KUKA KRL program: EPS_2_251245_SANMH3A_A_20250910013112.src

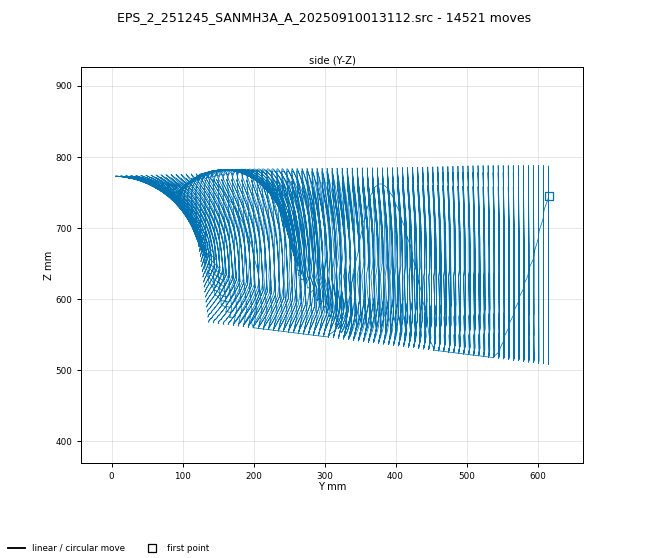
[picture p0: tool path of EPS_2_251245_SANMH3A_A_20250910013112.src, 14521 of 14523 moves have a stored position in this frame; points joined in program order, loops and branches not executed]
&ACCESS RVP
&REL 4
&COMMENT QRS 19112012
&PARAM EDITMASK = *
DEF PART()
EXT BAS (BAS_COMMAND :IN,REAL :IN )
INT I
BAS (#INITMOV,0 )

;KUKA QRS Post kuka4.cps  Date:22-06-2017 !

File_ID=2817

QRS_PRE_INIT()

;Init var - Until changes are made in qrs_pre_init
Outlet_Square_prg=0
Inlet_1_Square_prg=0
Inlet_2_Square_prg=0
Inlet_3_Square_prg=0
Inlet_4_Square_prg=0
Inlet_5_Square_prg=0

Outlet_1={X 0.000, Y 519.160, Z 687.500, B 0.000, E1 0.000 }
Inlet_1={X 0.000, Y 520.240, Z 710.500, B 0.000, E1 90.000 }
Inlet_2={X 0.000, Y 521.300, Z 657.500, B 0.000, E1 180.000 }
Outlet_1_type=201
Inlet_1_type=135
Inlet_2_type=201
;QRS#1=Sidecore dimensions
;QRS#2=200-8" PVC SDR 35
;QRS#3=135-5" PVC SDR 28
;QRS#4=200-8" PVC SDR 35
;QRS#5=
;QRS#6=
;QRS#7=
;QRS#8=
;QRS#9=12-08 PSX
;QRS#10=8-11 PSX
;QRS#11=12-08 PSX
;QRS#12=
;QRS#13=
;QRS#14=
;QRS#15=
;QRS#16=1220x127x1067 3,5'
;QRS#17=EPS Height
;QRS#18=788
;QRS#19=*
;QRS#20= UPDATED VERSION 22-06-2017
;QRS#21=*
Outlet_Square=0100
Inlet_1_Square=070
Inlet_2_Square=0100
Inlet_3_Square=0
Inlet_4_Square=0
Inlet_5_Square=0
Mill_Square=1
Outlet_Square_Prg=204
Inlet_1_Square_prg=202
Inlet_2_Square_prg=204

QRS_INIT()

$ADVANCE=5

; T1
PTP {E1 173.419,E2 173.419}
PTP {X 0,Y 615.493,A -85,B 0,C 180,E1 173.419,E2 173.419,E3 0,E4 0,E5 0,E6 0}
QRS_SPEED_INIT()
LIN {X 0,Y 615.493,Z 745.39,A -85,B 0,C 180,E1 173.419,E2 173.419,E3 0,E4 0,E5 0,E6 0} C_VEL
LIN {X 0,Y 615.498,Z 736.605,A -85,B 0,C 180,E1 172.784,E2 172.784} C_VEL
LIN {X 0,Y 615.5,Z 727.686,A -85,B 0,C 180,E1 172.29,E2 172.29} C_VEL
LIN {X 0,Y 615.493,Z 717.685,A -85,B 0,C 180,E1 171.877,E2 171.877} C_VEL
LIN {X 0,Y 615.488,Z 709.508,A -85,B 0,C 180,E1 171.629,E2 171.629} C_VEL
LIN {X 0,Y 615.491,Z 700.427,A -85,B 0,C 180,E1 171.443,E2 171.443} C_VEL
LIN {X 0,Y 615.487,Z 631.25,A -85,B 0,C 180,E1 170.615,E2 170.615} C_VEL
LIN {X 0,Y 615.498,Z 629.569,A -85,B 0,C 180,E1 170.47,E2 170.47} C_VEL
LIN {X 0,Y 615.491,Z 604.096,A -85,B 0,C 180,E1 167.47,E2 167.47} C_VEL
LIN {X 0,Y 615.496,Z 580.016,A -85,B 0,C 180,E1 164.605,E2 164.605} C_VEL
LIN {X 0,Y 615.48,Z 556.069,A -85,B 0,C 180,E1 161.719,E2 161.719} C_VEL
LIN {X 0,Y 615.495,Z 533.177,A -85,B 0,C 180,E1 158.919,E2 158.919} C_VEL
LIN {X 0,Y 615.496,Z 511.475,A -85,B 0,C 180,E1 156.217,E2 156.217} C_VEL
LIN {X 0,Y 615.495,Z 507.92,A -85,B 0,C 180,E1 155.728,E2 155.728} C_VEL
LIN {X 0,Y 615.497,Z 507.698,A -85,B 0,C 180,E1 153.556,E2 153.556} C_VEL
LIN {X 0,Y 615.49,Z 507.693,A -85,B 0,C 180,E1 151.342,E2 151.342} C_VEL
LIN {X 0,Y 615.477,Z 507.686,A -85,B 0,C 180,E1 148.916,E2 148.916} C_VEL
LIN {X 0,Y 615.485,Z 507.682,A -85,B 0,C 180,E1 146.467,E2 146.467} C_VEL
LIN {X 0,Y 615.489,Z 507.701,A -85,B 0,C 180,E1 143.575,E2 143.575} C_VEL
LIN {X 0,Y 615.479,Z 507.687,A -85,B 0,C 180,E1 140.939,E2 140.939} C_VEL
LIN {X 0,Y 615.482,Z 507.683,A -85,B 0,C 180,E1 138.525,E2 138.525} C_VEL
LIN {X 0,Y 615.485,Z 507.691,A -85,B 0,C 180,E1 135.85,E2 135.85} C_VEL
LIN {X 0,Y 615.485,Z 507.689,A -85,B 0,C 180,E1 133.047,E2 133.047} C_VEL
LIN {X 0,Y 615.478,Z 507.684,A -85,B 0,C 180,E1 130.608,E2 130.608} C_VEL
LIN {X 0,Y 615.489,Z 507.685,A -85,B 0,C 180,E1 128.012,E2 128.012} C_VEL
LIN {X 0,Y 615.488,Z 507.695,A -85,B 0,C 180,E1 125.616,E2 125.616} C_VEL
LIN {X 0,Y 615.492,Z 507.696,A -85,B 0,C 180,E1 123.236,E2 123.236} C_VEL
LIN {X 0,Y 615.479,Z 507.69,A -85,B 0,C 180,E1 120.921,E2 120.921} C_VEL
LIN {X 0,Y 615.481,Z 507.683,A -85,B 0,C 180,E1 118.449,E2 118.449} C_VEL
LIN {X 0,Y 615.484,Z 507.69,A -85,B 0,C 180,E1 115.716,E2 115.716} C_VEL
LIN {X 0,Y 615.48,Z 507.689,A -85,B 0,C 180,E1 112.845,E2 112.845} C_VEL
LIN {X 0,Y 615.493,Z 507.682,A -85,B 0,C 180,E1 110.033,E2 110.033} C_VEL
LIN {X 0,Y 615.498,Z 507.867,A -85,B 0,C 180,E1 109.208,E2 109.208} C_VEL
LIN {X 0,Y 615.49,Z 524.635,A -85,B 0,C 180,E1 106.431,E2 106.431} C_VEL
LIN {X 0,Y 615.487,Z 541.428,A -85,B 0,C 180,E1 103.706,E2 103.706} C_VEL
LIN {X 0,Y 615.484,Z 547.062,A -85,B 0,C 180,E1 102.845,E2 102.845} C_VEL
LIN {X 0,Y 615.481,Z 549.379,A -85,B 0,C 180,E1 102.782,E2 102.782} C_VEL
LIN {X 0,Y 615.497,Z 653.612,A -85,B 0,C 180,E1 101.548,E2 101.548} C_VEL
LIN {X 0,Y 615.498,Z 666.203,A -85,B 0,C 180,E1 101.277,E2 101.277} C_VEL
LIN {X 0,Y 615.497,Z 679.523,A -85,B 0,C 180,E1 100.845,E2 100.845} C_VEL
LIN {X 0,Y 615.495,Z 690.554,A -85,B 0,C 180,E1 100.361,E2 100.361} C_VEL
LIN {X 0,Y 615.489,Z 702.297,A -85,B 0,C 180,E1 99.697,E2 99.697} C_VEL
LIN {X 0,Y 615.499,Z 712.761,A -85,B 0,C 180,E1 98.951,E2 98.951} C_VEL
LIN {X 0,Y 615.498,Z 721.325,A -85,B 0,C 180,E1 98.206,E2 98.206} C_VEL
LIN {X 0,Y 615.497,Z 729.204,A -85,B 0,C 180,E1 97.381,E2 97.381} C_VEL
LIN {X 0,Y 615.497,Z 736.895,A -85,B 0,C 180,E1 96.393,E2 96.393} C_VEL
LIN {X 0,Y 615.497,Z 743.955,A -85,B 0,C 180,E1 95.242,E2 95.242} C_VEL
LIN {X 0,Y 615.494,Z 748.655,A -85,B 0,C 180,E1 94.257,E2 94.257} C_VEL
LIN {X 0,Y 615.494,Z 752.253,A -85,B 0,C 180,E1 93.273,E2 93.273} C_VEL
LIN {X 0,Y 615.496,Z 754.113,A -85,B 0,C 180,E1 92.618,E2 92.618} C_VEL
LIN {X 0,Y 615.498,Z 755.532,A -85,B 0,C 180,E1 91.964,E2 91.964} C_VEL
LIN {X 0,Y 615.496,Z 757.141,A -85,B 0,C 180,E1 90.655,E2 90.655} C_VEL
LIN {X 0,Y 615.495,Z 757.384,A -85,B 0,C 180,E1 90.001,E2 90.001} C_VEL
LIN {X 0,Y 615.495,Z 757.206,A -85,B 0,C 180,E1 89.346,E2 89.346} C_VEL
LIN {X 0,Y 615.499,Z 755.683,A -85,B 0,C 180,E1 88.038,E2 88.038} C_VEL
LIN {X 0,Y 615.498,Z 754.343,A -85,B 0,C 180,E1 87.383,E2 87.383} C_VEL
LIN {X 0,Y 615.496,Z 751.496,A -85,B 0,C 180,E1 86.4,E2 86.4} C_VEL
LIN {X 0,Y 615.498,Z 747.637,A -85,B 0,C 180,E1 85.416,E2 85.416} C_VEL
LIN {X 0,Y 615.498,Z 742.655,A -85,B 0,C 180,E1 84.431,E2 84.431} C_VEL
LIN {X 0,Y 615.496,Z 736.208,A -85,B 0,C 180,E1 83.418,E2 83.418} C_VEL
LIN {X 0,Y 615.497,Z 728.543,A -85,B 0,C 180,E1 82.455,E2 82.455} C_VEL
LIN {X 0,Y 615.498,Z 718.766,A -85,B 0,C 180,E1 81.464,E2 81.464} C_VEL
LIN {X 0,Y 615.498,Z 708.502,A -85,B 0,C 180,E1 80.636,E2 80.636} C_VEL
LIN {X 0,Y 615.495,Z 696.941,A -85,B 0,C 180,E1 79.889,E2 79.889} C_VEL
LIN {X 0,Y 615.497,Z 685.031,A -85,B 0,C 180,E1 79.291,E2 79.291} C_VEL
LIN {X 0,Y 615.497,Z 672.179,A -85,B 0,C 180,E1 78.808,E2 78.808} C_VEL
LIN {X 0,Y 615.497,Z 659.587,A -85,B 0,C 180,E1 78.474,E2 78.474} C_VEL
LIN {X 0,Y 615.498,Z 646.491,A -85,B 0,C 180,E1 78.265,E2 78.265} C_VEL
LIN {X 0,Y 615.487,Z 547.562,A -85,B 0,C 180,E1 77.093,E2 77.093} C_VEL
LIN {X 0,Y 615.486,Z 546.205,A -85,B 0,C 180,E1 76.967,E2 76.967} C_VEL
LIN {X 0,Y 615.486,Z 528.418,A -85,B 0,C 180,E1 74.096,E2 74.096} C_VEL
LIN {X 0,Y 615.496,Z 510.642,A -85,B 0,C 180,E1 71.182,E2 71.182} C_VEL
LIN {X 0,Y 615.493,Z 507.774,A -85,B 0,C 180,E1 70.663,E2 70.663} C_VEL
LIN {X 0,Y 615.494,Z 507.681,A -85,B 0,C 180,E1 67.865,E2 67.865} C_VEL
LIN {X 0,Y 615.488,Z 507.689,A -85,B 0,C 180,E1 65.009,E2 65.009} C_VEL
LIN {X 0,Y 615.488,Z 507.686,A -85,B 0,C 180,E1 62.086,E2 62.086} C_VEL
LIN {X 0,Y 615.499,Z 507.68,A -85,B 0,C 180,E1 59.841,E2 59.841} C_VEL
LIN {X 0,Y 615.481,Z 507.683,A -85,B 0,C 180,E1 57.543,E2 57.543} C_VEL
LIN {X 0,Y 615.478,Z 507.687,A -85,B 0,C 180,E1 55.185,E2 55.185} C_VEL
LIN {X 0,Y 615.496,Z 507.694,A -85,B 0,C 180,E1 52.759,E2 52.759} C_VEL
LIN {X 0,Y 615.492,Z 507.683,A -85,B 0,C 180,E1 49.911,E2 49.911} C_VEL
LIN {X 0,Y 615.49,Z 507.681,A -85,B 0,C 180,E1 47.648,E2 47.648} C_VEL
LIN {X 0,Y 615.482,Z 507.691,A -85,B 0,C 180,E1 44.932,E2 44.932} C_VEL
LIN {X 0,Y 615.483,Z 507.689,A -85,B 0,C 180,E1 42.081,E2 42.081} C_VEL
LIN {X 0,Y 615.498,Z 507.68,A -85,B 0,C 180,E1 39.75,E2 39.75} C_VEL
LIN {X 0,Y 615.48,Z 507.691,A -85,B 0,C 180,E1 36.937,E2 36.937} C_VEL
LIN {X 0,Y 615.494,Z 507.695,A -85,B 0,C 180,E1 34.703,E2 34.703} C_VEL
LIN {X 0,Y 615.486,Z 507.682,A -85,B 0,C 180,E1 31.686,E2 31.686} C_VEL
LIN {X 0,Y 615.482,Z 507.683,A -85,B 0,C 180,E1 29.407,E2 29.407} C_VEL
LIN {X 0,Y 615.478,Z 507.689,A -85,B 0,C 180,E1 27.045,E2 27.045} C_VEL
LIN {X 0,Y 615.486,Z 507.695,A -85,B 0,C 180,E1 24.272,E2 24.272} C_VEL
LIN {X 0,Y 615.486,Z 507.682,A -85,B 0,C 180,E1 21.432,E2 21.432} C_VEL
LIN {X 0,Y 615.495,Z 507.697,A -85,B 0,C 180,E1 18.61,E2 18.61} C_VEL
LIN {X 0,Y 615.483,Z 507.686,A -85,B 0,C 180,E1 15.905,E2 15.905} C_VEL
LIN {X 0,Y 615.478,Z 507.685,A -85,B 0,C 180,E1 13.202,E2 13.202} C_VEL
LIN {X 0,Y 615.494,Z 507.699,A -85,B 0,C 180,E1 10.527,E2 10.527} C_VEL
LIN {X 0,Y 615.482,Z 507.687,A -85,B 0,C 180,E1 7.876,E2 7.876} C_VEL
LIN {X 0,Y 615.481,Z 507.684,A -85,B 0,C 180,E1 5.241,E2 5.241} C_VEL
LIN {X 0,Y 615.491,Z 507.696,A -85,B 0,C 180,E1 2.618,E2 2.618} C_VEL
LIN {X 0,Y 615.479,Z 507.69,A -85,B 0,C 180,E1 0,E2 0} C_VEL
LIN {X 0,Y 615.491,Z 507.681,A -85,B 0,C 180,E1 -2.618,E2 -2.618} C_VEL
LIN {X 0,Y 615.477,Z 507.694,A -85,B 0,C 180,E1 -5.241,E2 -5.241} C_VEL
LIN {X 0,Y 615.482,Z 507.694,A -85,B 0,C 180,E1 -7.876,E2 -7.876} C_VEL
LIN {X 0,Y 615.489,Z 507.681,A -85,B 0,C 180,E1 -10.527,E2 -10.527} C_VEL
LIN {X 0,Y 615.478,Z 507.692,A -85,B 0,C 180,E1 -13.201,E2 -13.201} C_VEL
LIN {X 0,Y 615.481,Z 507.694,A -85,B 0,C 180,E1 -15.905,E2 -15.905} C_VEL
LIN {X 0,Y 615.49,Z 507.681,A -85,B 0,C 180,E1 -18.646,E2 -18.646} C_VEL
LIN {X 0,Y 615.486,Z 507.696,A -85,B 0,C 180,E1 -21.432,E2 -21.432} C_VEL
LIN {X 0,Y 615.478,Z 507.686,A -85,B 0,C 180,E1 -24.272,E2 -24.272} C_VEL
LIN {X 0,Y 615.478,Z 507.687,A -85,B 0,C 180,E1 -27.045,E2 -27.045} C_VEL
LIN {X 0,Y 615.488,Z 507.697,A -85,B 0,C 180,E1 -29.797,E2 -29.797} C_VEL
LIN {X 0,Y 615.484,Z 507.683,A -85,B 0,C 180,E1 -32.458,E2 -32.458} C_VEL
LIN {X 0,Y 615.491,Z 507.681,A -85,B 0,C 180,E1 -34.815,E2 -34.815} C_VEL
LIN {X 0,Y 615.476,Z 507.692,A -85,B 0,C 180,E1 -37.243,E2 -37.243} C_VEL
LIN {X 0,Y 615.478,Z 507.691,A -85,B 0,C 180,E1 -40.089,E2 -40.089} C_VEL
LIN {X 0,Y 615.478,Z 507.686,A -85,B 0,C 180,E1 -42.354,E2 -42.354} C_VEL
LIN {X 0,Y 615.482,Z 507.686,A -85,B 0,C 180,E1 -45.069,E2 -45.069} C_VEL
LIN {X 0,Y 615.488,Z 507.694,A -85,B 0,C 180,E1 -47.92,E2 -47.92} C_VEL
LIN {X 0,Y 615.477,Z 507.688,A -85,B 0,C 180,E1 -50.25,E2 -50.25} C_VEL
LIN {X 0,Y 615.484,Z 507.685,A -85,B 0,C 180,E1 -53.064,E2 -53.064} C_VEL
LIN {X 0,Y 615.487,Z 507.693,A -85,B 0,C 180,E1 -55.979,E2 -55.979} C_VEL
LIN {X 0,Y 615.476,Z 507.688,A -85,B 0,C 180,E1 -58.315,E2 -58.315} C_VEL
LIN {X 0,Y 615.478,Z 507.684,A -85,B 0,C 180,E1 -60.594,E2 -60.594} C_VEL
LIN {X 0,Y 615.492,Z 507.682,A -85,B 0,C 180,E1 -62.955,E2 -62.955} C_VEL
LIN {X 0,Y 615.493,Z 507.701,A -85,B 0,C 180,E1 -65.729,E2 -65.729} C_VEL
LIN {X 0,Y 615.493,Z 507.862,A -85,B 0,C 180,E1 -67.812,E2 -67.812} C_VEL
LIN {X 0,Y 615.498,Z 515.503,A -85,B 0,C 180,E1 -68.92,E2 -68.92} C_VEL
LIN {X 0,Y 615.486,Z 535.766,A -85,B 0,C 180,E1 -71.719,E2 -71.719} C_VEL
LIN {X 0,Y 615.477,Z 555.728,A -85,B 0,C 180,E1 -74.435,E2 -74.435} C_VEL
LIN {X 0,Y 615.498,Z 575.424,A -85,B 0,C 180,E1 -77.073,E2 -77.073} C_VEL
LIN {X 0,Y 615.495,Z 576.565,A -85,B 0,C 180,E1 -77.135,E2 -77.135} C_VEL
LIN {X 0,Y 615.496,Z 683.866,A -85,B 0,C 180,E1 -78.412,E2 -78.412} C_VEL
LIN {X 0,Y 615.498,Z 696.367,A -85,B 0,C 180,E1 -78.683,E2 -78.683} C_VEL
LIN {X 0,Y 615.496,Z 709.503,A -85,B 0,C 180,E1 -79.109,E2 -79.109} C_VEL
LIN {X 0,Y 615.487,Z 721.49,A -85,B 0,C 180,E1 -79.64,E2 -79.64} C_VEL
LIN {X 0,Y 615.482,Z 733.006,A -85,B 0,C 180,E1 -80.304,E2 -80.304} C_VEL
LIN {X 0,Y 615.499,Z 743.349,A -85,B 0,C 180,E1 -81.051,E2 -81.051} C_VEL
LIN {X 0,Y 615.497,Z 751.819,A -85,B 0,C 180,E1 -81.795,E2 -81.795} C_VEL
LIN {X 0,Y 615.498,Z 759.612,A -85,B 0,C 180,E1 -82.62,E2 -82.62} C_VEL
LIN {X 0,Y 615.496,Z 767.207,A -85,B 0,C 180,E1 -83.609,E2 -83.609} C_VEL
LIN {X 0,Y 615.498,Z 774.208,A -85,B 0,C 180,E1 -84.76,E2 -84.76} C_VEL
LIN {X 0,Y 615.493,Z 778.854,A -85,B 0,C 180,E1 -85.744,E2 -85.744} C_VEL
LIN {X 0,Y 615.495,Z 782.4,A -85,B 0,C 180,E1 -86.728,E2 -86.728} C_VEL
LIN {X 0,Y 615.497,Z 784.234,A -85,B 0,C 180,E1 -87.383,E2 -87.383} C_VEL
LIN {X 0,Y 615.496,Z 785.609,A -85,B 0,C 180,E1 -88.038,E2 -88.038} C_VEL
LIN {X 0,Y 615.496,Z 787.174,A -85,B 0,C 180,E1 -89.346,E2 -89.346} C_VEL
LIN {X 0,Y 615.494,Z 787.389,A -85,B 0,C 180,E1 -90.001,E2 -90.001} C_VEL
LIN {X 0,Y 615.496,Z 786.579,A -85,B 0,C 180,E1 -91.309,E2 -91.309} C_VEL
LIN {X 0,Y 615.496,Z 785.607,A -85,B 0,C 180,E1 -91.964,E2 -91.964} C_VEL
LIN {X 0,Y 615.497,Z 784.231,A -85,B 0,C 180,E1 -92.618,E2 -92.618} C_VEL
LIN {X 0,Y 615.496,Z 781.348,A -85,B 0,C 180,E1 -93.601,E2 -93.601} C_VEL
LIN {X 0,Y 615.498,Z 777.439,A -85,B 0,C 180,E1 -94.585,E2 -94.585} C_VEL
LIN {X 0,Y 615.499,Z 772.402,A -85,B 0,C 180,E1 -95.57,E2 -95.57} C_VEL
LIN {X 0,Y 615.497,Z 765.869,A -85,B 0,C 180,E1 -96.583,E2 -96.583} C_VEL
LIN {X 0,Y 615.497,Z 758.128,A -85,B 0,C 180,E1 -97.546,E2 -97.546} C_VEL
LIN {X 0,Y 615.498,Z 750.039,A -85,B 0,C 180,E1 -98.372,E2 -98.372} C_VEL
LIN {X 0,Y 615.499,Z 740.16,A -85,B 0,C 180,E1 -99.199,E2 -99.199} C_VEL
LIN {X 0,Y 615.483,Z 728.973,A -85,B 0,C 180,E1 -99.946,E2 -99.946} C_VEL
LIN {X 0,Y 615.488,Z 718.011,A -85,B 0,C 180,E1 -100.527,E2 -100.527} C_VEL
LIN {X 0,Y 615.499,Z 705.408,A -85,B 0,C 180,E1 -101.043,E2 -101.043} C_VEL
LIN {X 0,Y 615.498,Z 693.04,A -85,B 0,C 180,E1 -101.402,E2 -101.402} C_VEL
LIN {X 0,Y 615.496,Z 679.426,A -85,B 0,C 180,E1 -101.652,E2 -101.652} C_VEL
LIN {X 0,Y 615.494,Z 576.521,A -85,B 0,C 180,E1 -102.866,E2 -102.866} C_VEL
LIN {X 0,Y 615.497,Z 575.219,A -85,B 0,C 180,E1 -102.95,E2 -102.95} C_VEL
LIN {X 0,Y 615.479,Z 554.462,A -85,B 0,C 180,E1 -105.736,E2 -105.736} C_VEL
LIN {X 0,Y 615.493,Z 534.577,A -85,B 0,C 180,E1 -108.444,E2 -108.444} C_VEL
LIN {X 0,Y 615.497,Z 514.235,A -85,B 0,C 180,E1 -111.256,E2 -111.256} C_VEL
LIN {X 0,Y 615.493,Z 507.859,A -85,B 0,C 180,E1 -112.189,E2 -112.189} C_VEL
LIN {X 0,Y 615.49,Z 507.683,A -85,B 0,C 180,E1 -114.992,E2 -114.992} C_VEL
LIN {X 0,Y 615.483,Z 507.694,A -85,B 0,C 180,E1 -117.916,E2 -117.916} C_VEL
LIN {X 0,Y 615.499,Z 507.7,A -85,B 0,C 180,E1 -120.16,E2 -120.16} C_VEL
LIN {X 0,Y 615.481,Z 507.693,A -85,B 0,C 180,E1 -122.458,E2 -122.458} C_VEL
LIN {X 0,Y 615.478,Z 507.686,A -85,B 0,C 180,E1 -124.816,E2 -124.816} C_VEL
LIN {X 0,Y 615.492,Z 507.682,A -85,B 0,C 180,E1 -127.242,E2 -127.242} C_VEL
LIN {X 0,Y 615.497,Z 507.699,A -85,B 0,C 180,E1 -130.09,E2 -130.09} C_VEL
LIN {X 0,Y 615.49,Z 507.691,A -85,B 0,C 180,E1 -132.353,E2 -132.353} C_VEL
LIN {X 0,Y 615.481,Z 507.684,A -85,B 0,C 180,E1 -135.07,E2 -135.07} C_VEL
LIN {X 0,Y 615.494,Z 507.701,A -85,B 0,C 180,E1 -137.92,E2 -137.92} C_VEL
LIN {X 0,Y 615.499,Z 507.689,A -85,B 0,C 180,E1 -140.251,E2 -140.251} C_VEL
LIN {X 0,Y 615.479,Z 507.685,A -85,B 0,C 180,E1 -143.065,E2 -143.065} C_VEL
LIN {X 0,Y 615.492,Z 507.685,A -85,B 0,C 180,E1 -145.299,E2 -145.299} C_VEL
LIN {X 0,Y 615.495,Z 507.695,A -85,B 0,C 180,E1 -147.669,E2 -147.669} C_VEL
LIN {X 0,Y 615.482,Z 507.684,A -85,B 0,C 180,E1 -150.593,E2 -150.593} C_VEL
LIN {X 0,Y 615.478,Z 507.685,A -85,B 0,C 180,E1 -152.957,E2 -152.957} C_VEL
LIN {X 0,Y 615.495,Z 507.779,A -85,B 0,C 180,E1 -155.728,E2 -155.728} C_VEL
LIN {X 0,Y 615.495,Z 508.503,A -85,B 0,C 180,E1 -155.925,E2 -155.925} C_VEL
LIN {X 0,Y 615.486,Z 529.607,A -85,B 0,C 180,E1 -158.568,E2 -158.568} C_VEL
LIN {X 0,Y 615.495,Z 552.652,A -85,B 0,C 180,E1 -161.394,E2 -161.394} C_VEL
LIN {X 0,Y 615.488,Z 576.429,A -85,B 0,C 180,E1 -164.265,E2 -164.265} C_VEL
LIN {X 0,Y 615.483,Z 600.512,A -85,B 0,C 180,E1 -167.134,E2 -167.134} C_VEL
LIN {X 0,Y 615.488,Z 624.553,A -85,B 0,C 180,E1 -169.972,E2 -169.972} C_VEL
LIN {X 0,Y 615.484,Z 630.725,A -85,B 0,C 180,E1 -170.677,E2 -170.677} C_VEL
LIN {X 0,Y 615.481,Z 633.272,A -85,B 0,C 180,E1 -170.739,E2 -170.739} C_VEL
LIN {X 0,Y 615.491,Z 701.268,A -85,B 0,C 180,E1 -171.546,E2 -171.546} C_VEL
LIN {X 0,Y 615.492,Z 710.869,A -85,B 0,C 180,E1 -171.753,E2 -171.753} C_VEL
LIN {X 0,Y 615.496,Z 721.984,A -85,B 0,C 180,E1 -172.124,E2 -172.124} C_VEL
LIN {X 0,Y 615.499,Z 730.71,A -85,B 0,C 180,E1 -172.537,E2 -172.537} C_VEL
LIN {X 0,Y 615.494,Z 738.777,A -85,B 0,C 180,E1 -173.022,E2 -173.022} C_VEL
LIN {X 0,Y 615.497,Z 746.596,A -85,B 0,C 180,E1 -173.608,E2 -173.608} C_VEL
LIN {X 0,Y 615.499,Z 755.222,A -85,B 0,C 180,E1 -174.43,E2 -174.43} C_VEL
LIN {X 0,Y 615.497,Z 760.635,A -85,B 0,C 180,E1 -175.087,E2 -175.087} C_VEL
LIN {X 0,Y 615.493,Z 765.091,A -85,B 0,C 180,E1 -175.744,E2 -175.744} C_VEL
LIN {X 0,Y 615.494,Z 770.241,A -85,B 0,C 180,E1 -176.727,E2 -176.727} C_VEL
LIN {X 0,Y 615.497,Z 772.819,A -85,B 0,C 180,E1 -177.382,E2 -177.382} C_VEL
LIN {X 0,Y 615.49,Z 774.795,A -85,B 0,C 180,E1 -178.037,E2 -178.037} C_VEL
LIN {X 0,Y 615.491,Z 776.209,A -85,B 0,C 180,E1 -178.691,E2 -178.691} C_VEL
LIN {X 0,Y 615.49,Z 777.08,A -85,B 0,C 180,E1 -179.346,E2 -179.346} C_VEL
LIN {X 0,Y 615.492,Z 777.384,A -85,B 0,C 180,E1 -180,E2 -180} C_VEL
LIN {X 0,Y 615.493,Z 777.125,A -85,B 0,C 180,E1 -180.654,E2 -180.654} C_VEL
LIN {X 0,Y 615.496,Z 776.335,A -85,B 0,C 180,E1 -181.309,E2 -181.309} C_VEL
LIN {X 0,Y 615.49,Z 775.012,A -85,B 0,C 180,E1 -181.963,E2 -181.963} C_VEL
LIN {X 0,Y 615.494,Z 771.997,A -85,B 0,C 180,E1 -182.945,E2 -182.945} C_VEL
LIN {X 0,Y 615.495,Z 767.512,A -85,B 0,C 180,E1 -183.928,E2 -183.928} C_VEL
LIN {X 0,Y 615.494,Z 762.444,A -85,B 0,C 180,E1 -184.749,E2 -184.749} C_VEL
LIN {X 0,Y 615.499,Z 755.994,A -85,B 0,C 180,E1 -185.57,E2 -185.57} C_VEL
LIN {X 0,Y 615.496,Z 747.698,A -85,B 0,C 180,E1 -186.392,E2 -186.392} C_VEL
LIN {X 0,Y 615.493,Z 745.39,A -85,B 0,C 180,E1 -186.581,E2 -186.581} C_VEL
LIN {X 0,Y 614.822,Z 740.973,A -85,B 0,C 180,E1 -186.938,E2 -186.938} C_VEL
LIN {X 0,Y 611.962,Z 733.336,A -85,B 0,C 180,E1 -187.479,E2 -187.479} C_VEL
LIN {X 0,Y 609.578,Z 726.893,A -85,B 0,C 180,E1 -187.852,E2 -187.852} C_VEL
LIN {X 0,Y 608.569,Z 721.652,A -85,B 0,C 180,E1 -188.089,E2 -188.089} C_VEL
LIN {X 0,Y 608.497,Z 719.824,A -85,B 0,C 180,E1 -188.157,E2 -188.157} C_VEL
LIN {X 0,Y 608.479,Z 709.982,A -85,B 0,C 180,E1 -188.468,E2 -188.468} C_VEL
LIN {X 0,Y 608.513,Z 701.083,A -85,B 0,C 180,E1 -188.656,E2 -188.656} C_VEL
LIN {X 0,Y 608.491,Z 631.493,A -85,B 0,C 180,E1 -189.494,E2 -189.494} C_VEL
LIN {X 0,Y 608.468,Z 629.82,A -85,B 0,C 180,E1 -189.641,E2 -189.641} C_VEL
LIN {X 0,Y 608.488,Z 605.66,A -85,B 0,C 180,E1 -192.507,E2 -192.507} C_VEL
LIN {X 0,Y 608.486,Z 582.92,A -85,B 0,C 180,E1 -195.234,E2 -195.234} C_VEL
LIN {X 0,Y 608.542,Z 560.179,A -85,B 0,C 180,E1 -197.995,E2 -197.995} C_VEL
LIN {X 0,Y 608.591,Z 537.585,A -85,B 0,C 180,E1 -200.781,E2 -200.781} C_VEL
LIN {X 0,Y 608.623,Z 514.694,A -85,B 0,C 180,E1 -203.658,E2 -203.658} C_VEL
LIN {X 0,Y 608.508,Z 508.929,A -85,B 0,C 180,E1 -204.414,E2 -204.414} C_VEL
LIN {X 0,Y 608.451,Z 508.688,A -85,B 0,C 180,E1 -205.301,E2 -205.301} C_VEL
LIN {X 0,Y 608.447,Z 508.688,A -85,B 0,C 180,E1 -207.518,E2 -207.518} C_VEL
LIN {X 0,Y 608.47,Z 508.688,A -85,B 0,C 180,E1 -209.971,E2 -209.971} C_VEL
LIN {X 0,Y 608.457,Z 508.69,A -85,B 0,C 180,E1 -212.88,E2 -212.88} C_VEL
LIN {X 0,Y 608.449,Z 508.688,A -85,B 0,C 180,E1 -215.277,E2 -215.277} C_VEL
LIN {X 0,Y 608.468,Z 508.692,A -85,B 0,C 180,E1 -218.24,E2 -218.24} C_VEL
LIN {X 0,Y 608.454,Z 508.695,A -85,B 0,C 180,E1 -220.329,E2 -220.329} C_VEL
LIN {X 0,Y 608.447,Z 508.691,A -85,B 0,C 180,E1 -222.961,E2 -222.961} C_VEL
LIN {X 0,Y 608.462,Z 508.686,A -85,B 0,C 180,E1 -225.736,E2 -225.736} C_VEL
LIN {X 0,Y 608.468,Z 508.694,A -85,B 0,C 180,E1 -228.658,E2 -228.658} C_VEL
LIN {X 0,Y 608.467,Z 508.685,A -85,B 0,C 180,E1 -231.411,E2 -231.411} C_VEL
LIN {X 0,Y 608.45,Z 508.689,A -85,B 0,C 180,E1 -233.954,E2 -233.954} C_VEL
LIN {X 0,Y 608.471,Z 508.69,A -85,B 0,C 180,E1 -236.329,E2 -236.329} C_VEL
LIN {X 0,Y 608.452,Z 508.696,A -85,B 0,C 180,E1 -238.732,E2 -238.732} C_VEL
LIN {X 0,Y 608.468,Z 508.686,A -85,B 0,C 180,E1 -241.382,E2 -241.382} C_VEL
LIN {X 0,Y 608.442,Z 508.689,A -85,B 0,C 180,E1 -243.964,E2 -243.964} C_VEL
LIN {X 0,Y 608.471,Z 508.687,A -85,B 0,C 180,E1 -246.155,E2 -246.155} C_VEL
LIN {X 0,Y 608.455,Z 508.693,A -85,B 0,C 180,E1 -249.018,E2 -249.018} C_VEL
LIN {X 0,Y 608.49,Z 508.912,A -85,B 0,C 180,E1 -250.737,E2 -250.737} C_VEL
LIN {X 0,Y 608.479,Z 523.776,A -85,B 0,C 180,E1 -253.216,E2 -253.216} C_VEL
LIN {X 0,Y 608.48,Z 540.657,A -85,B 0,C 180,E1 -255.98,E2 -255.98} C_VEL
LIN {X 0,Y 608.497,Z 547.132,A -85,B 0,C 180,E1 -257.005,E2 -257.005} C_VEL
LIN {X 0,Y 608.573,Z 549.46,A -85,B 0,C 180,E1 -257.07,E2 -257.07} C_VEL
LIN {X 0,Y 608.557,Z 653.765,A -85,B 0,C 180,E1 -258.319,E2 -258.319} C_VEL
LIN {X 0,Y 608.539,Z 667.097,A -85,B 0,C 180,E1 -258.614,E2 -258.614} C_VEL
LIN {X 0,Y 608.529,Z 680.348,A -85,B 0,C 180,E1 -259.054,E2 -259.054} C_VEL
LIN {X 0,Y 608.505,Z 692.358,A -85,B 0,C 180,E1 -259.603,E2 -259.603} C_VEL
LIN {X 0,Y 608.502,Z 703.782,A -85,B 0,C 180,E1 -260.275,E2 -260.275} C_VEL
LIN {X 0,Y 608.474,Z 714.077,A -85,B 0,C 180,E1 -261.029,E2 -261.029} C_VEL
LIN {X 0,Y 608.464,Z 723.344,A -85,B 0,C 180,E1 -261.865,E2 -261.865} C_VEL
LIN {X 0,Y 608.467,Z 732.319,A -85,B 0,C 180,E1 -262.867,E2 -262.867} C_VEL
LIN {X 0,Y 608.444,Z 739.552,A -85,B 0,C 180,E1 -263.866,E2 -263.866} C_VEL
LIN {X 0,Y 608.462,Z 744.431,A -85,B 0,C 180,E1 -264.698,E2 -264.698} C_VEL
LIN {X 0,Y 608.439,Z 749.176,A -85,B 0,C 180,E1 -265.694,E2 -265.694} C_VEL
LIN {X 0,Y 608.425,Z 752.81,A -85,B 0,C 180,E1 -266.688,E2 -266.688} C_VEL
LIN {X 0,Y 608.425,Z 754.689,A -85,B 0,C 180,E1 -267.351,E2 -267.351} C_VEL
LIN {X 0,Y 608.443,Z 756.126,A -85,B 0,C 180,E1 -268.014,E2 -268.014} C_VEL
LIN {X 0,Y 608.439,Z 757.751,A -85,B 0,C 180,E1 -269.338,E2 -269.338} C_VEL
LIN {X 0,Y 608.435,Z 757.995,A -85,B 0,C 180,E1 -269.999,E2 -269.999} C_VEL
LIN {X 0,Y 608.438,Z 757.815,A -85,B 0,C 180,E1 -270.661,E2 -270.661} C_VEL
LIN {X 0,Y 608.444,Z 756.277,A -85,B 0,C 180,E1 -271.985,E2 -271.985} C_VEL
LIN {X 0,Y 608.426,Z 754.92,A -85,B 0,C 180,E1 -272.648,E2 -272.648} C_VEL
LIN {X 0,Y 608.449,Z 752.044,A -85,B 0,C 180,E1 -273.642,E2 -273.642} C_VEL
LIN {X 0,Y 608.433,Z 748.145,A -85,B 0,C 180,E1 -274.637,E2 -274.637} C_VEL
LIN {X 0,Y 608.449,Z 743.115,A -85,B 0,C 180,E1 -275.634,E2 -275.634} C_VEL
LIN {X 0,Y 608.441,Z 736.799,A -85,B 0,C 180,E1 -276.632,E2 -276.632} C_VEL
LIN {X 0,Y 608.475,Z 728.884,A -85,B 0,C 180,E1 -277.632,E2 -277.632} C_VEL
LIN {X 0,Y 608.472,Z 719.043,A -85,B 0,C 180,E1 -278.635,E2 -278.635} C_VEL
LIN {X 0,Y 608.48,Z 708.723,A -85,B 0,C 180,E1 -279.473,E2 -279.473} C_VEL
LIN {X 0,Y 608.491,Z 697.111,A -85,B 0,C 180,E1 -280.228,E2 -280.228} C_VEL
LIN {X 0,Y 608.529,Z 685.86,A -85,B 0,C 180,E1 -280.803,E2 -280.803} C_VEL
LIN {X 0,Y 608.538,Z 674.279,A -85,B 0,C 180,E1 -281.257,E2 -281.257} C_VEL
LIN {X 0,Y 608.539,Z 660.59,A -85,B 0,C 180,E1 -281.638,E2 -281.638} C_VEL
LIN {X 0,Y 608.572,Z 648.34,A -85,B 0,C 180,E1 -281.849,E2 -281.849} C_VEL
LIN {X 0,Y 608.53,Z 547.571,A -85,B 0,C 180,E1 -283.057,E2 -283.057} C_VEL
LIN {X 0,Y 608.481,Z 546.355,A -85,B 0,C 180,E1 -283.185,E2 -283.185} C_VEL
LIN {X 0,Y 608.49,Z 528.524,A -85,B 0,C 180,E1 -286.092,E2 -286.092} C_VEL
LIN {X 0,Y 608.511,Z 510.696,A -85,B 0,C 180,E1 -289.042,E2 -289.042} C_VEL
LIN {X 0,Y 608.481,Z 508.781,A -85,B 0,C 180,E1 -289.393,E2 -289.393} C_VEL
LIN {X 0,Y 608.477,Z 508.69,A -85,B 0,C 180,E1 -291.69,E2 -291.69} C_VEL
LIN {X 0,Y 608.455,Z 508.687,A -85,B 0,C 180,E1 -294.57,E2 -294.57} C_VEL
LIN {X 0,Y 608.484,Z 508.691,A -85,B 0,C 180,E1 -297.208,E2 -297.208} C_VEL
LIN {X 0,Y 608.471,Z 508.687,A -85,B 0,C 180,E1 -299.972,E2 -299.972} C_VEL
LIN {X 0,Y 608.457,Z 508.686,A -85,B 0,C 180,E1 -302.521,E2 -302.521} C_VEL
LIN {X 0,Y 608.471,Z 508.688,A -85,B 0,C 180,E1 -304.908,E2 -304.908} C_VEL
LIN {X 0,Y 608.474,Z 508.69,A -85,B 0,C 180,E1 -307.745,E2 -307.745} C_VEL
LIN {X 0,Y 608.451,Z 508.687,A -85,B 0,C 180,E1 -310.329,E2 -310.329} C_VEL
LIN {X 0,Y 608.485,Z 508.692,A -85,B 0,C 180,E1 -313.31,E2 -313.31} C_VEL
LIN {X 0,Y 608.468,Z 508.686,A -85,B 0,C 180,E1 -316.13,E2 -316.13} C_VEL
LIN {X 0,Y 608.449,Z 508.689,A -85,B 0,C 180,E1 -318.823,E2 -318.823} C_VEL
LIN {X 0,Y 608.466,Z 508.696,A -85,B 0,C 180,E1 -321.412,E2 -321.412} C_VEL
LIN {X 0,Y 608.474,Z 508.687,A -85,B 0,C 180,E1 -323.949,E2 -323.949} C_VEL
LIN {X 0,Y 608.463,Z 508.686,A -85,B 0,C 180,E1 -326.329,E2 -326.329} C_VEL
LIN {X 0,Y 608.471,Z 508.685,A -85,B 0,C 180,E1 -328.727,E2 -328.727} C_VEL
LIN {X 0,Y 608.476,Z 508.693,A -85,B 0,C 180,E1 -331.377,E2 -331.377} C_VEL
LIN {X 0,Y 608.476,Z 508.684,A -85,B 0,C 180,E1 -334.276,E2 -334.276} C_VEL
LIN {X 0,Y 608.448,Z 508.689,A -85,B 0,C 180,E1 -336.876,E2 -336.876} C_VEL
LIN {X 0,Y 608.463,Z 508.693,A -85,B 0,C 180,E1 -339.726,E2 -339.726} C_VEL
LIN {X 0,Y 608.445,Z 508.688,A -85,B 0,C 180,E1 -342.523,E2 -342.523} C_VEL
LIN {X 0,Y 608.477,Z 508.69,A -85,B 0,C 180,E1 -345.279,E2 -345.279} C_VEL
LIN {X 0,Y 608.459,Z 508.689,A -85,B 0,C 180,E1 -348,E2 -348} C_VEL
LIN {X 0,Y 608.463,Z 508.686,A -85,B 0,C 180,E1 -350.694,E2 -350.694} C_VEL
LIN {X 0,Y 608.469,Z 508.693,A -85,B 0,C 180,E1 -353.367,E2 -353.367} C_VEL
LIN {X 0,Y 608.448,Z 508.69,A -85,B 0,C 180,E1 -356.026,E2 -356.026} C_VEL
LIN {X 0,Y 608.468,Z 508.685,A -85,B 0,C 180,E1 -358.676,E2 -358.676} C_VEL
LIN {X 0,Y 608.468,Z 508.692,A -85,B 0,C 180,E1 -361.324,E2 -361.324} C_VEL
LIN {X 0,Y 608.45,Z 508.691,A -85,B 0,C 180,E1 -363.974,E2 -363.974} C_VEL
LIN {X 0,Y 608.469,Z 508.685,A -85,B 0,C 180,E1 -366.633,E2 -366.633} C_VEL
LIN {X 0,Y 608.462,Z 508.692,A -85,B 0,C 180,E1 -369.306,E2 -369.306} C_VEL
LIN {X 0,Y 608.458,Z 508.69,A -85,B 0,C 180,E1 -372,E2 -372} C_VEL
LIN {X 0,Y 608.473,Z 508.684,A -85,B 0,C 180,E1 -374.721,E2 -374.721} C_VEL
LIN {X 0,Y 608.445,Z 508.696,A -85,B 0,C 180,E1 -377.477,E2 -377.477} C_VEL
LIN {X 0,Y 608.458,Z 508.688,A -85,B 0,C 180,E1 -380.274,E2 -380.274} C_VEL
LIN {X 0,Y 608.451,Z 508.687,A -85,B 0,C 180,E1 -382.477,E2 -382.477} C_VEL
LIN {X 0,Y 608.451,Z 508.692,A -85,B 0,C 180,E1 -385.301,E2 -385.301} C_VEL
LIN {X 0,Y 608.443,Z 508.697,A -85,B 0,C 180,E1 -387.518,E2 -387.518} C_VEL
LIN {X 0,Y 608.464,Z 508.69,A -85,B 0,C 180,E1 -389.973,E2 -389.973} C_VEL
LIN {X 0,Y 608.458,Z 508.686,A -85,B 0,C 180,E1 -392.524,E2 -392.524} C_VEL
LIN {X 0,Y 608.451,Z 508.692,A -85,B 0,C 180,E1 -395.277,E2 -395.277} C_VEL
LIN {X 0,Y 608.461,Z 508.696,A -85,B 0,C 180,E1 -397.747,E2 -397.747} C_VEL
LIN {X 0,Y 608.446,Z 508.689,A -85,B 0,C 180,E1 -400.33,E2 -400.33} C_VEL
LIN {X 0,Y 608.468,Z 508.689,A -85,B 0,C 180,E1 -403.31,E2 -403.31} C_VEL
LIN {X 0,Y 608.469,Z 508.688,A -85,B 0,C 180,E1 -406.132,E2 -406.132} C_VEL
LIN {X 0,Y 608.455,Z 508.687,A -85,B 0,C 180,E1 -408.825,E2 -408.825} C_VEL
LIN {X 0,Y 608.468,Z 508.691,A -85,B 0,C 180,E1 -411.413,E2 -411.413} C_VEL
LIN {X 0,Y 608.474,Z 508.691,A -85,B 0,C 180,E1 -413.951,E2 -413.951} C_VEL
LIN {X 0,Y 608.463,Z 508.687,A -85,B 0,C 180,E1 -416.33,E2 -416.33} C_VEL
LIN {X 0,Y 608.477,Z 508.683,A -85,B 0,C 180,E1 -418.728,E2 -418.728} C_VEL
LIN {X 0,Y 608.47,Z 508.69,A -85,B 0,C 180,E1 -421.381,E2 -421.381} C_VEL
LIN {X 0,Y 608.441,Z 508.695,A -85,B 0,C 180,E1 -423.965,E2 -423.965} C_VEL
LIN {X 0,Y 608.466,Z 508.69,A -85,B 0,C 180,E1 -426.156,E2 -426.156} C_VEL
LIN {X 0,Y 608.503,Z 508.815,A -85,B 0,C 180,E1 -427.686,E2 -427.686} C_VEL
LIN {X 0,Y 608.567,Z 518.026,A -85,B 0,C 180,E1 -429.023,E2 -429.023} C_VEL
LIN {X 0,Y 608.521,Z 536.986,A -85,B 0,C 180,E1 -431.667,E2 -431.667} C_VEL
LIN {X 0,Y 608.487,Z 557.065,A -85,B 0,C 180,E1 -434.424,E2 -434.424} C_VEL
LIN {X 0,Y 608.498,Z 575.741,A -85,B 0,C 180,E1 -436.942,E2 -436.942} C_VEL
LIN {X 0,Y 608.587,Z 577.99,A -85,B 0,C 180,E1 -437.008,E2 -437.008} C_VEL
LIN {X 0,Y 608.547,Z 683.984,A -85,B 0,C 180,E1 -438.277,E2 -438.277} C_VEL
LIN {X 0,Y 608.547,Z 697.24,A -85,B 0,C 180,E1 -438.573,E2 -438.573} C_VEL
LIN {X 0,Y 608.544,Z 710.338,A -85,B 0,C 180,E1 -439.009,E2 -439.009} C_VEL
LIN {X 0,Y 608.506,Z 721.648,A -85,B 0,C 180,E1 -439.52,E2 -439.52} C_VEL
LIN {X 0,Y 608.472,Z 733.207,A -85,B 0,C 180,E1 -440.192,E2 -440.192} C_VEL
LIN {X 0,Y 608.485,Z 743.602,A -85,B 0,C 180,E1 -440.946,E2 -440.946} C_VEL
LIN {X 0,Y 608.475,Z 752.119,A -85,B 0,C 180,E1 -441.699,E2 -441.699} C_VEL
LIN {X 0,Y 608.471,Z 759.966,A -85,B 0,C 180,E1 -442.535,E2 -442.535} C_VEL
LIN {X 0,Y 608.46,Z 767.289,A -85,B 0,C 180,E1 -443.485,E2 -443.485} C_VEL
LIN {X 0,Y 608.45,Z 772.869,A -85,B 0,C 180,E1 -444.366,E2 -444.366} C_VEL
LIN {X 0,Y 608.432,Z 777.953,A -85,B 0,C 180,E1 -445.363,E2 -445.363} C_VEL
LIN {X 0,Y 608.449,Z 781.898,A -85,B 0,C 180,E1 -446.358,E2 -446.358} C_VEL
LIN {X 0,Y 608.425,Z 784.811,A -85,B 0,C 180,E1 -447.352,E2 -447.352} C_VEL
LIN {X 0,Y 608.441,Z 786.202,A -85,B 0,C 180,E1 -448.015,E2 -448.015} C_VEL
LIN {X 0,Y 608.438,Z 787.784,A -85,B 0,C 180,E1 -449.339,E2 -449.339} C_VEL
LIN {X 0,Y 608.434,Z 788,A -85,B 0,C 180,E1 -450.001,E2 -450.001} C_VEL
LIN {X 0,Y 608.448,Z 787.183,A -85,B 0,C 180,E1 -451.324,E2 -451.324} C_VEL
LIN {X 0,Y 608.441,Z 786.2,A -85,B 0,C 180,E1 -451.986,E2 -451.986} C_VEL
LIN {X 0,Y 608.425,Z 784.808,A -85,B 0,C 180,E1 -452.649,E2 -452.649} C_VEL
LIN {X 0,Y 608.449,Z 781.894,A -85,B 0,C 180,E1 -453.643,E2 -453.643} C_VEL
LIN {X 0,Y 608.432,Z 777.948,A -85,B 0,C 180,E1 -454.638,E2 -454.638} C_VEL
LIN {X 0,Y 608.437,Z 771.873,A -85,B 0,C 180,E1 -455.801,E2 -455.801} C_VEL
LIN {X 0,Y 608.462,Z 765.231,A -85,B 0,C 180,E1 -456.8,E2 -456.8} C_VEL
LIN {X 0,Y 608.456,Z 756.984,A -85,B 0,C 180,E1 -457.801,E2 -457.801} C_VEL
LIN {X 0,Y 608.472,Z 748.53,A -85,B 0,C 180,E1 -458.636,E2 -458.636} C_VEL
LIN {X 0,Y 608.475,Z 738.083,A -85,B 0,C 180,E1 -459.474,E2 -459.474} C_VEL
LIN {X 0,Y 608.482,Z 727.746,A -85,B 0,C 180,E1 -460.145,E2 -460.145} C_VEL
LIN {X 0,Y 608.522,Z 716.231,A -85,B 0,C 180,E1 -460.741,E2 -460.741} C_VEL
LIN {X 0,Y 608.541,Z 703.863,A -85,B 0,C 180,E1 -461.225,E2 -461.225} C_VEL
LIN {X 0,Y 608.55,Z 690.417,A -85,B 0,C 180,E1 -461.597,E2 -461.597} C_VEL
LIN {X 0,Y 608.553,Z 678.043,A -85,B 0,C 180,E1 -461.808,E2 -461.808} C_VEL
LIN {X 0,Y 608.56,Z 576.537,A -85,B 0,C 180,E1 -463.015,E2 -463.015} C_VEL
LIN {X 0,Y 608.489,Z 575.346,A -85,B 0,C 180,E1 -463.101,E2 -463.101} C_VEL
LIN {X 0,Y 608.494,Z 554.537,A -85,B 0,C 180,E1 -465.921,E2 -465.921} C_VEL
LIN {X 0,Y 608.52,Z 535.793,A -85,B 0,C 180,E1 -468.499,E2 -468.499} C_VEL
LIN {X 0,Y 608.574,Z 515.499,A -85,B 0,C 180,E1 -471.332,E2 -471.332} C_VEL
LIN {X 0,Y 608.503,Z 508.811,A -85,B 0,C 180,E1 -472.315,E2 -472.315} C_VEL
LIN {X 0,Y 608.458,Z 508.692,A -85,B 0,C 180,E1 -474.571,E2 -474.571} C_VEL
LIN {X 0,Y 608.482,Z 508.684,A -85,B 0,C 180,E1 -477.207,E2 -477.207} C_VEL
LIN {X 0,Y 608.467,Z 508.692,A -85,B 0,C 180,E1 -479.971,E2 -479.971} C_VEL
LIN {X 0,Y 608.456,Z 508.688,A -85,B 0,C 180,E1 -482.88,E2 -482.88} C_VEL
LIN {X 0,Y 608.438,Z 508.689,A -85,B 0,C 180,E1 -485.278,E2 -485.278} C_VEL
LIN {X 0,Y 608.474,Z 508.69,A -85,B 0,C 180,E1 -487.746,E2 -487.746} C_VEL
LIN {X 0,Y 608.453,Z 508.693,A -85,B 0,C 180,E1 -490.329,E2 -490.329} C_VEL
LIN {X 0,Y 608.485,Z 508.684,A -85,B 0,C 180,E1 -493.31,E2 -493.31} C_VEL
LIN {X 0,Y 608.476,Z 508.692,A -85,B 0,C 180,E1 -496.131,E2 -496.131} C_VEL
LIN {X 0,Y 608.449,Z 508.688,A -85,B 0,C 180,E1 -498.823,E2 -498.823} C_VEL
LIN {X 0,Y 608.469,Z 508.688,A -85,B 0,C 180,E1 -501.412,E2 -501.412} C_VEL
LIN {X 0,Y 608.481,Z 508.693,A -85,B 0,C 180,E1 -503.951,E2 -503.951} C_VEL
LIN {X 0,Y 608.469,Z 508.688,A -85,B 0,C 180,E1 -506.33,E2 -506.33} C_VEL
LIN {X 0,Y 608.447,Z 508.688,A -85,B 0,C 180,E1 -508.733,E2 -508.733} C_VEL
LIN {X 0,Y 608.479,Z 508.688,A -85,B 0,C 180,E1 -511.38,E2 -511.38} C_VEL
LIN {X 0,Y 608.478,Z 508.688,A -85,B 0,C 180,E1 -514.278,E2 -514.278} C_VEL
LIN {X 0,Y 608.472,Z 508.85,A -85,B 0,C 180,E1 -515.647,E2 -515.647} C_VEL
LIN {X 0,Y 608.64,Z 510.764,A -85,B 0,C 180,E1 -515.933,E2 -515.933} C_VEL
LIN {X 0,Y 608.567,Z 532.453,A -85,B 0,C 180,E1 -518.668,E2 -518.668} C_VEL
LIN {X 0,Y 608.556,Z 555.346,A -85,B 0,C 180,E1 -521.503,E2 -521.503} C_VEL
LIN {X 0,Y 608.526,Z 579.333,A -85,B 0,C 180,E1 -524.424,E2 -524.424} C_VEL
LIN {X 0,Y 608.487,Z 603.485,A -85,B 0,C 180,E1 -527.323,E2 -527.323} C_VEL
LIN {X 0,Y 608.485,Z 627.638,A -85,B 0,C 180,E1 -530.191,E2 -530.191} C_VEL
LIN {X 0,Y 608.475,Z 631.327,A -85,B 0,C 180,E1 -530.589,E2 -530.589} C_VEL
LIN {X 0,Y 608.496,Z 701.992,A -85,B 0,C 180,E1 -531.448,E2 -531.448} C_VEL
LIN {X 0,Y 608.49,Z 712.974,A -85,B 0,C 180,E1 -531.699,E2 -531.699} C_VEL
LIN {X 0,Y 608.491,Z 722.376,A -85,B 0,C 180,E1 -532.033,E2 -532.033} C_VEL
LIN {X 0,Y 608.496,Z 731.1,A -85,B 0,C 180,E1 -532.451,E2 -532.451} C_VEL
LIN {X 0,Y 608.484,Z 739.323,A -85,B 0,C 180,E1 -532.951,E2 -532.951} C_VEL
LIN {X 0,Y 608.468,Z 746.573,A -85,B 0,C 180,E1 -533.497,E2 -533.497} C_VEL
LIN {X 0,Y 608.458,Z 754.158,A -85,B 0,C 180,E1 -534.199,E2 -534.199} C_VEL
LIN {X 0,Y 608.438,Z 761.126,A -85,B 0,C 180,E1 -535.03,E2 -535.03} C_VEL
LIN {X 0,Y 608.439,Z 765.61,A -85,B 0,C 180,E1 -535.694,E2 -535.694} C_VEL
LIN {X 0,Y 608.427,Z 770.798,A -85,B 0,C 180,E1 -536.689,E2 -536.689} C_VEL
LIN {X 0,Y 608.427,Z 773.397,A -85,B 0,C 180,E1 -537.352,E2 -537.352} C_VEL
LIN {X 0,Y 608.436,Z 775.387,A -85,B 0,C 180,E1 -538.014,E2 -538.014} C_VEL
LIN {X 0,Y 608.443,Z 776.812,A -85,B 0,C 180,E1 -538.676,E2 -538.676} C_VEL
LIN {X 0,Y 608.434,Z 777.688,A -85,B 0,C 180,E1 -539.338,E2 -539.338} C_VEL
LIN {X 0,Y 608.433,Z 777.995,A -85,B 0,C 180,E1 -540,E2 -540} C_VEL
LIN {X 0,Y 608.436,Z 777.736,A -85,B 0,C 180,E1 -540.662,E2 -540.662} C_VEL
LIN {X 0,Y 608.448,Z 776.94,A -85,B 0,C 180,E1 -541.324,E2 -541.324} C_VEL
LIN {X 0,Y 608.436,Z 775.604,A -85,B 0,C 180,E1 -541.986,E2 -541.986} C_VEL
LIN {X 0,Y 608.449,Z 772.563,A -85,B 0,C 180,E1 -542.98,E2 -542.98} C_VEL
LIN {X 0,Y 608.433,Z 768.043,A -85,B 0,C 180,E1 -543.974,E2 -543.974} C_VEL
LIN {X 0,Y 608.446,Z 762.94,A -85,B 0,C 180,E1 -544.804,E2 -544.804} C_VEL
LIN {X 0,Y 608.471,Z 756.451,A -85,B 0,C 180,E1 -545.634,E2 -545.634} C_VEL
LIN {X 0,Y 608.454,Z 749.215,A -85,B 0,C 180,E1 -546.372,E2 -546.372} C_VEL
LIN {X 0,Y 608.484,Z 740.637,A -85,B 0,C 180,E1 -547.049,E2 -547.049} C_VEL
LIN {X 0,Y 608.496,Z 732.703,A -85,B 0,C 180,E1 -547.549,E2 -547.549} C_VEL
LIN {X 0,Y 608.493,Z 724.373,A -85,B 0,C 180,E1 -547.967,E2 -547.967} C_VEL
LIN {X 0,Y 608.497,Z 719.824,A -85,B 0,C 180,E1 -548.157,E2 -548.157} C_VEL
LIN {X 0,Y 608.031,Z 714.298,A -85,B 0,C 180,E1 -548.356,E2 -548.356} C_VEL
LIN {X 0,Y 606.537,Z 708.846,A -85,B 0,C 180,E1 -548.531,E2 -548.531} C_VEL
LIN {X 0,Y 602.727,Z 697.882,A -85,B 0,C 180,E1 -548.792,E2 -548.792} C_VEL
LIN {X 0,Y 601.579,Z 692.158,A -85,B 0,C 180,E1 -548.878,E2 -548.878} C_VEL
LIN {X 0,Y 601.486,Z 690.208,A -85,B 0,C 180,E1 -548.903,E2 -548.903} C_VEL
LIN {X 0,Y 601.451,Z 631.474,A -85,B 0,C 180,E1 -549.606,E2 -549.606} C_VEL
LIN {X 0,Y 601.42,Z 629.816,A -85,B 0,C 180,E1 -549.755,E2 -549.755} C_VEL
LIN {X 0,Y 601.468,Z 605.655,A -85,B 0,C 180,E1 -552.656,E2 -552.656} C_VEL
LIN {X 0,Y 601.531,Z 581.494,A -85,B 0,C 180,E1 -555.588,E2 -555.588} C_VEL
LIN {X 0,Y 601.6,Z 557.295,A -85,B 0,C 180,E1 -558.567,E2 -558.567} C_VEL
LIN {X 0,Y 601.668,Z 534.589,A -85,B 0,C 180,E1 -561.409,E2 -561.409} C_VEL
LIN {X 0,Y 601.782,Z 514.689,A -85,B 0,C 180,E1 -563.943,E2 -563.943} C_VEL
LIN {X 0,Y 601.466,Z 509.836,A -85,B 0,C 180,E1 -564.599,E2 -564.599} C_VEL
LIN {X 0,Y 601.411,Z 509.57,A -85,B 0,C 180,E1 -564.878,E2 -564.878} C_VEL
LIN {X 0,Y 601.413,Z 509.565,A -85,B 0,C 180,E1 -567.361,E2 -567.361} C_VEL
LIN {X 0,Y 601.432,Z 509.568,A -85,B 0,C 180,E1 -570.149,E2 -570.149} C_VEL
LIN {X 0,Y 601.427,Z 509.568,A -85,B 0,C 180,E1 -572.716,E2 -572.716} C_VEL
LIN {X 0,Y 601.416,Z 509.565,A -85,B 0,C 180,E1 -575.114,E2 -575.114} C_VEL
LIN {X 0,Y 601.437,Z 509.561,A -85,B 0,C 180,E1 -577.419,E2 -577.419} C_VEL
LIN {X 0,Y 601.415,Z 509.566,A -85,B 0,C 180,E1 -579.995,E2 -579.995} C_VEL
LIN {X 0,Y 601.412,Z 509.571,A -85,B 0,C 180,E1 -582.671,E2 -582.671} C_VEL
LIN {X 0,Y 601.431,Z 509.561,A -85,B 0,C 180,E1 -585.482,E2 -585.482} C_VEL
LIN {X 0,Y 601.43,Z 509.57,A -85,B 0,C 180,E1 -588.407,E2 -588.407} C_VEL
LIN {X 0,Y 601.417,Z 509.568,A -85,B 0,C 180,E1 -590.873,E2 -590.873} C_VEL
LIN {X 0,Y 601.403,Z 509.565,A -85,B 0,C 180,E1 -593.417,E2 -593.417} C_VEL
LIN {X 0,Y 601.436,Z 509.563,A -85,B 0,C 180,E1 -596.064,E2 -596.064} C_VEL
LIN {X 0,Y 601.434,Z 509.571,A -85,B 0,C 180,E1 -598.544,E2 -598.544} C_VEL
LIN {X 0,Y 601.428,Z 509.563,A -85,B 0,C 180,E1 -601.373,E2 -601.373} C_VEL
LIN {X 0,Y 601.403,Z 509.565,A -85,B 0,C 180,E1 -603.636,E2 -603.636} C_VEL
LIN {X 0,Y 601.422,Z 509.572,A -85,B 0,C 180,E1 -606.589,E2 -606.589} C_VEL
LIN {X 0,Y 601.428,Z 509.565,A -85,B 0,C 180,E1 -609.478,E2 -609.478} C_VEL
LIN {X 0,Y 601.464,Z 509.728,A -85,B 0,C 180,E1 -610.636,E2 -610.636} C_VEL
LIN {X 0,Y 601.497,Z 523.779,A -85,B 0,C 180,E1 -613.016,E2 -613.016} C_VEL
LIN {X 0,Y 601.432,Z 541.227,A -85,B 0,C 180,E1 -615.906,E2 -615.906} C_VEL
LIN {X 0,Y 601.468,Z 547.142,A -85,B 0,C 180,E1 -616.85,E2 -616.85} C_VEL
LIN {X 0,Y 601.678,Z 549.505,A -85,B 0,C 180,E1 -616.919,E2 -616.919} C_VEL
LIN {X 0,Y 601.63,Z 653.795,A -85,B 0,C 180,E1 -618.182,E2 -618.182} C_VEL
LIN {X 0,Y 601.603,Z 667.117,A -85,B 0,C 180,E1 -618.481,E2 -618.481} C_VEL
LIN {X 0,Y 601.545,Z 679.482,A -85,B 0,C 180,E1 -618.892,E2 -618.892} C_VEL
LIN {X 0,Y 601.522,Z 690.737,A -85,B 0,C 180,E1 -619.396,E2 -619.396} C_VEL
LIN {X 0,Y 601.482,Z 702.514,A -85,B 0,C 180,E1 -620.075,E2 -620.075} C_VEL
LIN {X 0,Y 601.445,Z 713.026,A -85,B 0,C 180,E1 -620.838,E2 -620.838} C_VEL
LIN {X 0,Y 601.43,Z 721.634,A -85,B 0,C 180,E1 -621.6,E2 -621.6} C_VEL
LIN {X 0,Y 601.418,Z 729.564,A -85,B 0,C 180,E1 -622.445,E2 -622.445} C_VEL
LIN {X 0,Y 601.377,Z 736.886,A -85,B 0,C 180,E1 -623.393,E2 -623.393} C_VEL
LIN {X 0,Y 601.372,Z 742.609,A -85,B 0,C 180,E1 -624.298,E2 -624.298} C_VEL
LIN {X 0,Y 601.335,Z 747.751,A -85,B 0,C 180,E1 -625.307,E2 -625.307} C_VEL
LIN {X 0,Y 601.367,Z 751.741,A -85,B 0,C 180,E1 -626.314,E2 -626.314} C_VEL
LIN {X 0,Y 601.324,Z 754.691,A -85,B 0,C 180,E1 -627.32,E2 -627.32} C_VEL
LIN {X 0,Y 601.342,Z 756.126,A -85,B 0,C 180,E1 -627.99,E2 -627.99} C_VEL
LIN {X 0,Y 601.339,Z 757.752,A -85,B 0,C 180,E1 -629.33,E2 -629.33} C_VEL
LIN {X 0,Y 601.336,Z 757.995,A -85,B 0,C 180,E1 -629.999,E2 -629.999} C_VEL
LIN {X 0,Y 601.339,Z 757.815,A -85,B 0,C 180,E1 -630.669,E2 -630.669} C_VEL
LIN {X 0,Y 601.343,Z 756.277,A -85,B 0,C 180,E1 -632.009,E2 -632.009} C_VEL
LIN {X 0,Y 601.326,Z 754.918,A -85,B 0,C 180,E1 -632.679,E2 -632.679} C_VEL
LIN {X 0,Y 601.368,Z 752.042,A -85,B 0,C 180,E1 -633.685,E2 -633.685} C_VEL
LIN {X 0,Y 601.337,Z 748.143,A -85,B 0,C 180,E1 -634.692,E2 -634.692} C_VEL
LIN {X 0,Y 601.373,Z 743.113,A -85,B 0,C 180,E1 -635.7,E2 -635.7} C_VEL
LIN {X 0,Y 601.382,Z 736.796,A -85,B 0,C 180,E1 -636.711,E2 -636.711} C_VEL
LIN {X 0,Y 601.396,Z 728.879,A -85,B 0,C 180,E1 -637.723,E2 -637.723} C_VEL
LIN {X 0,Y 601.436,Z 719.037,A -85,B 0,C 180,E1 -638.737,E2 -638.737} C_VEL
LIN {X 0,Y 601.449,Z 708.717,A -85,B 0,C 180,E1 -639.584,E2 -639.584} C_VEL
LIN {X 0,Y 601.493,Z 697.102,A -85,B 0,C 180,E1 -640.348,E2 -640.348} C_VEL
LIN {X 0,Y 601.551,Z 685.849,A -85,B 0,C 180,E1 -640.93,E2 -640.93} C_VEL
LIN {X 0,Y 601.565,Z 673.343,A -85,B 0,C 180,E1 -641.419,E2 -641.419} C_VEL
LIN {X 0,Y 601.601,Z 660.568,A -85,B 0,C 180,E1 -641.775,E2 -641.775} C_VEL
LIN {X 0,Y 601.641,Z 648.301,A -85,B 0,C 180,E1 -641.987,E2 -641.987} C_VEL
LIN {X 0,Y 601.593,Z 548.393,A -85,B 0,C 180,E1 -643.189,E2 -643.189} C_VEL
LIN {X 0,Y 601.437,Z 546.958,A -85,B 0,C 180,E1 -643.257,E2 -643.257} C_VEL
LIN {X 0,Y 601.468,Z 529.569,A -85,B 0,C 180,E1 -646.111,E2 -646.111} C_VEL
LIN {X 0,Y 601.538,Z 511.741,A -85,B 0,C 180,E1 -649.094,E2 -649.094} C_VEL
LIN {X 0,Y 601.46,Z 509.632,A -85,B 0,C 180,E1 -649.496,E2 -649.496} C_VEL
LIN {X 0,Y 601.415,Z 509.566,A -85,B 0,C 180,E1 -651.958,E2 -651.958} C_VEL
LIN {X 0,Y 601.44,Z 509.561,A -85,B 0,C 180,E1 -654.293,E2 -654.293} C_VEL
LIN {X 0,Y 601.456,Z 509.564,A -85,B 0,C 180,E1 -657.11,E2 -657.11} C_VEL
LIN {X 0,Y 601.42,Z 509.573,A -85,B 0,C 180,E1 -659.392,E2 -659.392} C_VEL
LIN {X 0,Y 601.414,Z 509.569,A -85,B 0,C 180,E1 -661.725,E2 -661.725} C_VEL
LIN {X 0,Y 601.429,Z 509.563,A -85,B 0,C 180,E1 -664.117,E2 -664.117} C_VEL
LIN {X 0,Y 601.41,Z 509.564,A -85,B 0,C 180,E1 -666.581,E2 -666.581} C_VEL
LIN {X 0,Y 601.438,Z 509.57,A -85,B 0,C 180,E1 -669.535,E2 -669.535} C_VEL
LIN {X 0,Y 601.413,Z 509.564,A -85,B 0,C 180,E1 -672.59,E2 -672.59} C_VEL
LIN {X 0,Y 601.421,Z 509.563,A -85,B 0,C 180,E1 -674.534,E2 -674.534} C_VEL
LIN {X 0,Y 601.41,Z 509.575,A -85,B 0,C 180,E1 -677.408,E2 -677.408} C_VEL
LIN {X 0,Y 601.411,Z 509.566,A -85,B 0,C 180,E1 -680.005,E2 -680.005} C_VEL
LIN {X 0,Y 601.43,Z 509.562,A -85,B 0,C 180,E1 -682.617,E2 -682.617} C_VEL
LIN {X 0,Y 601.437,Z 509.565,A -85,B 0,C 180,E1 -685.069,E2 -685.069} C_VEL
LIN {X 0,Y 601.434,Z 509.572,A -85,B 0,C 180,E1 -687.484,E2 -687.484} C_VEL
LIN {X 0,Y 601.443,Z 509.565,A -85,B 0,C 180,E1 -689.847,E2 -689.847} C_VEL
LIN {X 0,Y 601.41,Z 509.564,A -85,B 0,C 180,E1 -692.636,E2 -692.636} C_VEL
LIN {X 0,Y 601.4,Z 509.57,A -85,B 0,C 180,E1 -695.121,E2 -695.121} C_VEL
LIN {X 0,Y 601.41,Z 509.573,A -85,B 0,C 180,E1 -697.393,E2 -697.393} C_VEL
LIN {X 0,Y 601.403,Z 509.566,A -85,B 0,C 180,E1 -700.19,E2 -700.19} C_VEL
LIN {X 0,Y 601.428,Z 509.565,A -85,B 0,C 180,E1 -703.014,E2 -703.014} C_VEL
LIN {X 0,Y 601.415,Z 509.568,A -85,B 0,C 180,E1 -705.907,E2 -705.907} C_VEL
LIN {X 0,Y 601.428,Z 509.562,A -85,B 0,C 180,E1 -708.542,E2 -708.542} C_VEL
LIN {X 0,Y 601.436,Z 509.567,A -85,B 0,C 180,E1 -711.262,E2 -711.262} C_VEL
LIN {X 0,Y 601.408,Z 509.568,A -85,B 0,C 180,E1 -713.963,E2 -713.963} C_VEL
LIN {X 0,Y 601.426,Z 509.562,A -85,B 0,C 180,E1 -716.65,E2 -716.65} C_VEL
LIN {X 0,Y 601.448,Z 509.566,A -85,B 0,C 180,E1 -719.33,E2 -719.33} C_VEL
LIN {X 0,Y 601.42,Z 509.566,A -85,B 0,C 180,E1 -722.009,E2 -722.009} C_VEL
LIN {X 0,Y 601.429,Z 509.562,A -85,B 0,C 180,E1 -724.692,E2 -724.692} C_VEL
LIN {X 0,Y 601.434,Z 509.569,A -85,B 0,C 180,E1 -727.385,E2 -727.385} C_VEL
LIN {X 0,Y 601.428,Z 509.564,A -85,B 0,C 180,E1 -730.095,E2 -730.095} C_VEL
LIN {X 0,Y 601.419,Z 509.564,A -85,B 0,C 180,E1 -732.828,E2 -732.828} C_VEL
LIN {X 0,Y 601.409,Z 509.575,A -85,B 0,C 180,E1 -735.591,E2 -735.591} C_VEL
LIN {X 0,Y 601.419,Z 509.564,A -85,B 0,C 180,E1 -738.392,E2 -738.392} C_VEL
LIN {X 0,Y 601.404,Z 509.569,A -85,B 0,C 180,E1 -741.239,E2 -741.239} C_VEL
LIN {X 0,Y 601.449,Z 509.562,A -85,B 0,C 180,E1 -744.141,E2 -744.141} C_VEL
LIN {X 0,Y 601.444,Z 509.562,A -85,B 0,C 180,E1 -747.112,E2 -747.112} C_VEL
LIN {X 0,Y 601.42,Z 509.57,A -85,B 0,C 180,E1 -749.393,E2 -749.393} C_VEL
LIN {X 0,Y 601.409,Z 509.574,A -85,B 0,C 180,E1 -751.727,E2 -751.727} C_VEL
LIN {X 0,Y 601.427,Z 509.565,A -85,B 0,C 180,E1 -754.119,E2 -754.119} C_VEL
LIN {X 0,Y 601.407,Z 509.564,A -85,B 0,C 180,E1 -756.583,E2 -756.583} C_VEL
LIN {X 0,Y 601.439,Z 509.569,A -85,B 0,C 180,E1 -759.537,E2 -759.537} C_VEL
LIN {X 0,Y 601.407,Z 509.564,A -85,B 0,C 180,E1 -762.591,E2 -762.591} C_VEL
LIN {X 0,Y 601.422,Z 509.57,A -85,B 0,C 180,E1 -765.483,E2 -765.483} C_VEL
LIN {X 0,Y 601.423,Z 509.564,A -85,B 0,C 180,E1 -768.407,E2 -768.407} C_VEL
LIN {X 0,Y 601.434,Z 509.561,A -85,B 0,C 180,E1 -770.876,E2 -770.876} C_VEL
LIN {X 0,Y 601.441,Z 509.571,A -85,B 0,C 180,E1 -773.735,E2 -773.735} C_VEL
LIN {X 0,Y 601.426,Z 509.562,A -85,B 0,C 180,E1 -776.687,E2 -776.687} C_VEL
LIN {X 0,Y 601.432,Z 509.56,A -85,B 0,C 180,E1 -779.06,E2 -779.06} C_VEL
LIN {X 0,Y 601.429,Z 509.567,A -85,B 0,C 180,E1 -781.374,E2 -781.374} C_VEL
LIN {X 0,Y 601.403,Z 509.575,A -85,B 0,C 180,E1 -783.637,E2 -783.637} C_VEL
LIN {X 0,Y 601.418,Z 509.566,A -85,B 0,C 180,E1 -786.59,E2 -786.59} C_VEL
LIN {X 0,Y 601.436,Z 509.666,A -85,B 0,C 180,E1 -787.526,E2 -787.526} C_VEL
LIN {X 0,Y 601.642,Z 511.745,A -85,B 0,C 180,E1 -787.872,E2 -787.872} C_VEL
LIN {X 0,Y 601.575,Z 531.879,A -85,B 0,C 180,E1 -790.73,E2 -790.73} C_VEL
LIN {X 0,Y 601.524,Z 551.5,A -85,B 0,C 180,E1 -793.469,E2 -793.469} C_VEL
LIN {X 0,Y 601.455,Z 572.349,A -85,B 0,C 180,E1 -796.337,E2 -796.337} C_VEL
LIN {X 0,Y 601.493,Z 576.035,A -85,B 0,C 180,E1 -796.809,E2 -796.809} C_VEL
LIN {X 0,Y 601.691,Z 579.779,A -85,B 0,C 180,E1 -796.878,E2 -796.878} C_VEL
LIN {X 0,Y 601.595,Z 683.984,A -85,B 0,C 180,E1 -798.14,E2 -798.14} C_VEL
LIN {X 0,Y 601.589,Z 697.24,A -85,B 0,C 180,E1 -798.439,E2 -798.439} C_VEL
LIN {X 0,Y 601.575,Z 709.667,A -85,B 0,C 180,E1 -798.855,E2 -798.855} C_VEL
LIN {X 0,Y 601.527,Z 721.647,A -85,B 0,C 180,E1 -799.397,E2 -799.397} C_VEL
LIN {X 0,Y 601.474,Z 733.209,A -85,B 0,C 180,E1 -800.076,E2 -800.076} C_VEL
LIN {X 0,Y 601.444,Z 743.603,A -85,B 0,C 180,E1 -800.84,E2 -800.84} C_VEL
LIN {X 0,Y 601.429,Z 752.119,A -85,B 0,C 180,E1 -801.601,E2 -801.601} C_VEL
LIN {X 0,Y 601.417,Z 759.966,A -85,B 0,C 180,E1 -802.446,E2 -802.446} C_VEL
LIN {X 0,Y 601.369,Z 767.228,A -85,B 0,C 180,E1 -803.398,E2 -803.398} C_VEL
LIN {X 0,Y 601.371,Z 772.87,A -85,B 0,C 180,E1 -804.3,E2 -804.3} C_VEL
LIN {X 0,Y 601.337,Z 777.953,A -85,B 0,C 180,E1 -805.308,E2 -805.308} C_VEL
LIN {X 0,Y 601.367,Z 781.898,A -85,B 0,C 180,E1 -806.315,E2 -806.315} C_VEL
LIN {X 0,Y 601.325,Z 784.811,A -85,B 0,C 180,E1 -807.321,E2 -807.321} C_VEL
LIN {X 0,Y 601.34,Z 786.203,A -85,B 0,C 180,E1 -807.991,E2 -807.991} C_VEL
LIN {X 0,Y 601.339,Z 787.784,A -85,B 0,C 180,E1 -809.331,E2 -809.331} C_VEL
LIN {X 0,Y 601.335,Z 788,A -85,B 0,C 180,E1 -810.001,E2 -810.001} C_VEL
LIN {X 0,Y 601.348,Z 787.183,A -85,B 0,C 180,E1 -811.34,E2 -811.34} C_VEL
LIN {X 0,Y 601.34,Z 786.201,A -85,B 0,C 180,E1 -812.01,E2 -812.01} C_VEL
LIN {X 0,Y 601.325,Z 784.807,A -85,B 0,C 180,E1 -812.68,E2 -812.68} C_VEL
LIN {X 0,Y 601.367,Z 781.894,A -85,B 0,C 180,E1 -813.686,E2 -813.686} C_VEL
LIN {X 0,Y 601.337,Z 777.948,A -85,B 0,C 180,E1 -814.693,E2 -814.693} C_VEL
LIN {X 0,Y 601.372,Z 771.873,A -85,B 0,C 180,E1 -815.87,E2 -815.87} C_VEL
LIN {X 0,Y 601.382,Z 765.231,A -85,B 0,C 180,E1 -816.88,E2 -816.88} C_VEL
LIN {X 0,Y 601.4,Z 756.984,A -85,B 0,C 180,E1 -817.893,E2 -817.893} C_VEL
LIN {X 0,Y 601.436,Z 748.53,A -85,B 0,C 180,E1 -818.738,E2 -818.738} C_VEL
LIN {X 0,Y 601.442,Z 738.085,A -85,B 0,C 180,E1 -819.586,E2 -819.586} C_VEL
LIN {X 0,Y 601.478,Z 727.748,A -85,B 0,C 180,E1 -820.265,E2 -820.265} C_VEL
LIN {X 0,Y 601.538,Z 716.888,A -85,B 0,C 180,E1 -820.836,E2 -820.836} C_VEL
LIN {X 0,Y 601.566,Z 704.361,A -85,B 0,C 180,E1 -821.341,E2 -821.341} C_VEL
LIN {X 0,Y 601.606,Z 691.331,A -85,B 0,C 180,E1 -821.712,E2 -821.712} C_VEL
LIN {X 0,Y 601.623,Z 678.043,A -85,B 0,C 180,E1 -821.946,E2 -821.946} C_VEL
LIN {X 0,Y 601.533,Z 576.525,A -85,B 0,C 180,E1 -823.17,E2 -823.17} C_VEL
LIN {X 0,Y 601.469,Z 575.346,A -85,B 0,C 180,E1 -823.257,E2 -823.257} C_VEL
LIN {X 0,Y 601.522,Z 553.278,A -85,B 0,C 180,E1 -826.285,E2 -826.285} C_VEL
LIN {X 0,Y 601.6,Z 533.129,A -85,B 0,C 180,E1 -829.093,E2 -829.093} C_VEL
LIN {X 0,Y 601.664,Z 512.98,A -85,B 0,C 180,E1 -831.95,E2 -831.95} C_VEL
LIN {X 0,Y 601.457,Z 509.737,A -85,B 0,C 180,E1 -832.447,E2 -832.447} C_VEL
LIN {X 0,Y 601.405,Z 509.567,A -85,B 0,C 180,E1 -834.879,E2 -834.879} C_VEL
LIN {X 0,Y 601.419,Z 509.564,A -85,B 0,C 180,E1 -837.363,E2 -837.363} C_VEL
LIN {X 0,Y 601.433,Z 509.572,A -85,B 0,C 180,E1 -840.164,E2 -840.164} C_VEL
LIN {X 0,Y 601.42,Z 509.565,A -85,B 0,C 180,E1 -842.715,E2 -842.715} C_VEL
LIN {X 0,Y 601.393,Z 509.567,A -85,B 0,C 180,E1 -845.111,E2 -845.111} C_VEL
LIN {X 0,Y 601.439,Z 509.562,A -85,B 0,C 180,E1 -847.419,E2 -847.419} C_VEL
LIN {X 0,Y 601.406,Z 509.575,A -85,B 0,C 180,E1 -849.996,E2 -849.996} C_VEL
LIN {X 0,Y 601.415,Z 509.565,A -85,B 0,C 180,E1 -852.67,E2 -852.67} C_VEL
LIN {X 0,Y 601.43,Z 509.565,A -85,B 0,C 180,E1 -855.482,E2 -855.482} C_VEL
LIN {X 0,Y 601.425,Z 509.566,A -85,B 0,C 180,E1 -858.407,E2 -858.407} C_VEL
LIN {X 0,Y 601.435,Z 509.562,A -85,B 0,C 180,E1 -860.875,E2 -860.875} C_VEL
LIN {X 0,Y 601.446,Z 509.569,A -85,B 0,C 180,E1 -863.734,E2 -863.734} C_VEL
LIN {X 0,Y 601.429,Z 509.563,A -85,B 0,C 180,E1 -866.686,E2 -866.686} C_VEL
LIN {X 0,Y 601.416,Z 509.565,A -85,B 0,C 180,E1 -869.058,E2 -869.058} C_VEL
LIN {X 0,Y 601.438,Z 509.566,A -85,B 0,C 180,E1 -871.373,E2 -871.373} C_VEL
LIN {X 0,Y 601.419,Z 509.571,A -85,B 0,C 180,E1 -874.132,E2 -874.132} C_VEL
LIN {X 0,Y 601.427,Z 509.694,A -85,B 0,C 180,E1 -875.444,E2 -875.444} C_VEL
LIN {X 0,Y 601.793,Z 512.571,A -85,B 0,C 180,E1 -875.874,E2 -875.874} C_VEL
LIN {X 0,Y 601.681,Z 535.299,A -85,B 0,C 180,E1 -878.771,E2 -878.771} C_VEL
LIN {X 0,Y 601.578,Z 558.028,A -85,B 0,C 180,E1 -881.613,E2 -881.613} C_VEL
LIN {X 0,Y 601.53,Z 580.758,A -85,B 0,C 180,E1 -884.412,E2 -884.412} C_VEL
LIN {X 0,Y 601.469,Z 604.91,A -85,B 0,C 180,E1 -887.344,E2 -887.344} C_VEL
LIN {X 0,Y 601.419,Z 629.063,A -85,B 0,C 180,E1 -890.245,E2 -890.245} C_VEL
LIN {X 0,Y 601.449,Z 631.334,A -85,B 0,C 180,E1 -890.479,E2 -890.479} C_VEL
LIN {X 0,Y 601.495,Z 702.059,A -85,B 0,C 180,E1 -891.348,E2 -891.348} C_VEL
LIN {X 0,Y 601.462,Z 712.986,A -85,B 0,C 180,E1 -891.601,E2 -891.601} C_VEL
LIN {X 0,Y 601.458,Z 722.399,A -85,B 0,C 180,E1 -891.939,E2 -891.939} C_VEL
LIN {X 0,Y 601.442,Z 731.119,A -85,B 0,C 180,E1 -892.362,E2 -892.362} C_VEL
LIN {X 0,Y 601.419,Z 739.34,A -85,B 0,C 180,E1 -892.868,E2 -892.868} C_VEL
LIN {X 0,Y 601.413,Z 746.875,A -85,B 0,C 180,E1 -893.444,E2 -893.444} C_VEL
LIN {X 0,Y 601.388,Z 754.166,A -85,B 0,C 180,E1 -894.131,E2 -894.131} C_VEL
LIN {X 0,Y 601.35,Z 761.135,A -85,B 0,C 180,E1 -894.971,E2 -894.971} C_VEL
LIN {X 0,Y 601.358,Z 765.618,A -85,B 0,C 180,E1 -895.643,E2 -895.643} C_VEL
LIN {X 0,Y 601.346,Z 770.805,A -85,B 0,C 180,E1 -896.65,E2 -896.65} C_VEL
LIN {X 0,Y 601.33,Z 773.405,A -85,B 0,C 180,E1 -897.32,E2 -897.32} C_VEL
LIN {X 0,Y 601.336,Z 775.391,A -85,B 0,C 180,E1 -897.991,E2 -897.991} C_VEL
LIN {X 0,Y 601.343,Z 776.818,A -85,B 0,C 180,E1 -898.661,E2 -898.661} C_VEL
LIN {X 0,Y 601.334,Z 777.69,A -85,B 0,C 180,E1 -899.33,E2 -899.33} C_VEL
LIN {X 0,Y 601.333,Z 777.996,A -85,B 0,C 180,E1 -900,E2 -900} C_VEL
LIN {X 0,Y 601.336,Z 777.74,A -85,B 0,C 180,E1 -900.67,E2 -900.67} C_VEL
LIN {X 0,Y 601.347,Z 776.944,A -85,B 0,C 180,E1 -901.339,E2 -901.339} C_VEL
LIN {X 0,Y 601.335,Z 775.605,A -85,B 0,C 180,E1 -902.009,E2 -902.009} C_VEL
LIN {X 0,Y 601.347,Z 772.567,A -85,B 0,C 180,E1 -903.015,E2 -903.015} C_VEL
LIN {X 0,Y 601.345,Z 768.045,A -85,B 0,C 180,E1 -904.021,E2 -904.021} C_VEL
LIN {X 0,Y 601.379,Z 762.942,A -85,B 0,C 180,E1 -904.86,E2 -904.86} C_VEL
LIN {X 0,Y 601.392,Z 756.453,A -85,B 0,C 180,E1 -905.701,E2 -905.701} C_VEL
LIN {X 0,Y 601.404,Z 748.484,A -85,B 0,C 180,E1 -906.512,E2 -906.512} C_VEL
LIN {X 0,Y 601.419,Z 740.638,A -85,B 0,C 180,E1 -907.132,E2 -907.132} C_VEL
LIN {X 0,Y 601.442,Z 732.702,A -85,B 0,C 180,E1 -907.638,E2 -907.638} C_VEL
LIN {X 0,Y 601.451,Z 724.375,A -85,B 0,C 180,E1 -908.061,E2 -908.061} C_VEL
LIN {X 0,Y 601.475,Z 714.481,A -85,B 0,C 180,E1 -908.441,E2 -908.441} C_VEL
LIN {X 0,Y 601.516,Z 703.678,A -85,B 0,C 180,E1 -908.715,E2 -908.715} C_VEL
LIN {X 0,Y 601.486,Z 690.208,A -85,B 0,C 180,E1 -908.903,E2 -908.903} C_VEL
LIN {X 0,Y 600.82,Z 684.39,A -85,B 0,C 180,E1 -908.981,E2 -908.981} C_VEL
LIN {X 0,Y 595.123,Z 665.654,A -85,B 0,C 180,E1 -909.292,E2 -909.292} C_VEL
LIN {X 0,Y 594.524,Z 659.837,A -85,B 0,C 180,E1 -909.371,E2 -909.371} C_VEL
LIN {X 0,Y 594.391,Z 631.455,A -85,B 0,C 180,E1 -909.722,E2 -909.722} C_VEL
LIN {X 0,Y 594.37,Z 629.811,A -85,B 0,C 180,E1 -909.872,E2 -909.872} C_VEL
LIN {X 0,Y 594.441,Z 605.651,A -85,B 0,C 180,E1 -912.808,E2 -912.808} C_VEL
LIN {X 0,Y 594.556,Z 581.489,A -85,B 0,C 180,E1 -915.776,E2 -915.776} C_VEL
LIN {X 0,Y 594.668,Z 557.635,A -85,B 0,C 180,E1 -918.748,E2 -918.748} C_VEL
LIN {X 0,Y 594.79,Z 534.585,A -85,B 0,C 180,E1 -921.669,E2 -921.669} C_VEL
LIN {X 0,Y 594.945,Z 514.684,A -85,B 0,C 180,E1 -924.236,E2 -924.236} C_VEL
LIN {X 0,Y 594.405,Z 510.636,A -85,B 0,C 180,E1 -924.818,E2 -924.818} C_VEL
LIN {X 0,Y 594.372,Z 510.443,A -85,B 0,C 180,E1 -927.523,E2 -927.523} C_VEL
LIN {X 0,Y 594.389,Z 510.449,A -85,B 0,C 180,E1 -930.328,E2 -930.328} C_VEL
LIN {X 0,Y 594.382,Z 510.443,A -85,B 0,C 180,E1 -932.95,E2 -932.95} C_VEL
LIN {X 0,Y 594.387,Z 510.439,A -85,B 0,C 180,E1 -935.407,E2 -935.407} C_VEL
LIN {X 0,Y 594.389,Z 510.441,A -85,B 0,C 180,E1 -937.941,E2 -937.941} C_VEL
LIN {X 0,Y 594.378,Z 510.444,A -85,B 0,C 180,E1 -940.822,E2 -940.822} C_VEL
LIN {X 0,Y 594.369,Z 510.44,A -85,B 0,C 180,E1 -943.3,E2 -943.3} C_VEL
LIN {X 0,Y 594.387,Z 510.443,A -85,B 0,C 180,E1 -946.159,E2 -946.159} C_VEL
LIN {X 0,Y 594.38,Z 510.441,A -85,B 0,C 180,E1 -949.178,E2 -949.178} C_VEL
LIN {X 0,Y 594.391,Z 510.441,A -85,B 0,C 180,E1 -952.059,E2 -952.059} C_VEL
LIN {X 0,Y 594.355,Z 510.452,A -85,B 0,C 180,E1 -954.676,E2 -954.676} C_VEL
LIN {X 0,Y 594.383,Z 510.443,A -85,B 0,C 180,E1 -957.088,E2 -957.088} C_VEL
LIN {X 0,Y 594.391,Z 510.439,A -85,B 0,C 180,E1 -959.672,E2 -959.672} C_VEL
LIN {X 0,Y 594.38,Z 510.449,A -85,B 0,C 180,E1 -962.539,E2 -962.539} C_VEL
LIN {X 0,Y 594.379,Z 510.448,A -85,B 0,C 180,E1 -964.807,E2 -964.807} C_VEL
LIN {X 0,Y 594.369,Z 510.444,A -85,B 0,C 180,E1 -967.265,E2 -967.265} C_VEL
LIN {X 0,Y 594.377,Z 510.444,A -85,B 0,C 180,E1 -969.946,E2 -969.946} C_VEL
LIN {X 0,Y 594.411,Z 510.631,A -85,B 0,C 180,E1 -970.554,E2 -970.554} C_VEL
LIN {X 0,Y 594.491,Z 521.686,A -85,B 0,C 180,E1 -972.454,E2 -972.454} C_VEL
LIN {X 0,Y 594.43,Z 538.458,A -85,B 0,C 180,E1 -975.274,E2 -975.274} C_VEL
LIN {X 0,Y 594.439,Z 547.151,A -85,B 0,C 180,E1 -976.692,E2 -976.692} C_VEL
LIN {X 0,Y 594.764,Z 549.55,A -85,B 0,C 180,E1 -976.765,E2 -976.765} C_VEL
LIN {X 0,Y 594.686,Z 653.825,A -85,B 0,C 180,E1 -978.042,E2 -978.042} C_VEL
LIN {X 0,Y 594.636,Z 667.138,A -85,B 0,C 180,E1 -978.344,E2 -978.344} C_VEL
LIN {X 0,Y 594.584,Z 680.361,A -85,B 0,C 180,E1 -978.794,E2 -978.794} C_VEL
LIN {X 0,Y 594.524,Z 692.379,A -85,B 0,C 180,E1 -979.355,E2 -979.355} C_VEL
LIN {X 0,Y 594.472,Z 703.801,A -85,B 0,C 180,E1 -980.043,E2 -980.043} C_VEL
LIN {X 0,Y 594.406,Z 714.093,A -85,B 0,C 180,E1 -980.815,E2 -980.815} C_VEL
LIN {X 0,Y 594.373,Z 723.354,A -85,B 0,C 180,E1 -981.671,E2 -981.671} C_VEL
LIN {X 0,Y 594.317,Z 732.328,A -85,B 0,C 180,E1 -982.696,E2 -982.696} C_VEL
LIN {X 0,Y 594.285,Z 738.854,A -85,B 0,C 180,E1 -983.612,E2 -983.612} C_VEL
LIN {X 0,Y 594.289,Z 744.438,A -85,B 0,C 180,E1 -984.571,E2 -984.571} C_VEL
LIN {X 0,Y 594.27,Z 749.181,A -85,B 0,C 180,E1 -985.591,E2 -985.591} C_VEL
LIN {X 0,Y 594.267,Z 752.815,A -85,B 0,C 180,E1 -986.609,E2 -986.609} C_VEL
LIN {X 0,Y 594.225,Z 754.693,A -85,B 0,C 180,E1 -987.288,E2 -987.288} C_VEL
LIN {X 0,Y 594.241,Z 756.127,A -85,B 0,C 180,E1 -987.966,E2 -987.966} C_VEL
LIN {X 0,Y 594.24,Z 757.753,A -85,B 0,C 180,E1 -989.322,E2 -989.322} C_VEL
LIN {X 0,Y 594.236,Z 757.996,A -85,B 0,C 180,E1 -989.999,E2 -989.999} C_VEL
LIN {X 0,Y 594.239,Z 757.815,A -85,B 0,C 180,E1 -990.677,E2 -990.677} C_VEL
LIN {X 0,Y 594.241,Z 756.276,A -85,B 0,C 180,E1 -992.033,E2 -992.033} C_VEL
LIN {X 0,Y 594.226,Z 754.917,A -85,B 0,C 180,E1 -992.711,E2 -992.711} C_VEL
LIN {X 0,Y 594.289,Z 752.04,A -85,B 0,C 180,E1 -993.729,E2 -993.729} C_VEL
LIN {X 0,Y 594.241,Z 748.141,A -85,B 0,C 180,E1 -994.748,E2 -994.748} C_VEL
LIN {X 0,Y 594.299,Z 743.11,A -85,B 0,C 180,E1 -995.768,E2 -995.768} C_VEL
LIN {X 0,Y 594.316,Z 736.792,A -85,B 0,C 180,E1 -996.791,E2 -996.791} C_VEL
LIN {X 0,Y 594.346,Z 728.874,A -85,B 0,C 180,E1 -997.815,E2 -997.815} C_VEL
LIN {X 0,Y 594.381,Z 719.03,A -85,B 0,C 180,E1 -998.841,E2 -998.841} C_VEL
LIN {X 0,Y 594.431,Z 708.712,A -85,B 0,C 180,E1 -999.699,E2 -999.699} C_VEL
LIN {X 0,Y 594.508,Z 697.091,A -85,B 0,C 180,E1 -1000.471,E2 -1000.471} C_VEL
LIN {X 0,Y 594.572,Z 685.156,A -85,B 0,C 180,E1 -1001.09,E2 -1001.09} C_VEL
LIN {X 0,Y 594.601,Z 673.401,A -85,B 0,C 180,E1 -1001.553,E2 -1001.553} C_VEL
LIN {X 0,Y 594.655,Z 660.546,A -85,B 0,C 180,E1 -1001.914,E2 -1001.914} C_VEL
LIN {X 0,Y 594.705,Z 648.262,A -85,B 0,C 180,E1 -1002.129,E2 -1002.129} C_VEL
LIN {X 0,Y 594.677,Z 549.212,A -85,B 0,C 180,E1 -1003.332,E2 -1003.332} C_VEL
LIN {X 0,Y 594.427,Z 547.208,A -85,B 0,C 180,E1 -1003.394,E2 -1003.394} C_VEL
LIN {X 0,Y 594.458,Z 530.615,A -85,B 0,C 180,E1 -1006.13,E2 -1006.13} C_VEL
LIN {X 0,Y 594.539,Z 513.222,A -85,B 0,C 180,E1 -1009.074,E2 -1009.074} C_VEL
LIN {X 0,Y 594.402,Z 510.515,A -85,B 0,C 180,E1 -1009.579,E2 -1009.579} C_VEL
LIN {X 0,Y 594.361,Z 510.443,A -85,B 0,C 180,E1 -1012.233,E2 -1012.233} C_VEL
LIN {X 0,Y 594.39,Z 510.439,A -85,B 0,C 180,E1 -1014.445,E2 -1014.445} C_VEL
LIN {X 0,Y 594.387,Z 510.44,A -85,B 0,C 180,E1 -1016.699,E2 -1016.699} C_VEL
LIN {X 0,Y 594.381,Z 510.444,A -85,B 0,C 180,E1 -1018.998,E2 -1018.998} C_VEL
LIN {X 0,Y 594.392,Z 510.445,A -85,B 0,C 180,E1 -1021.644,E2 -1021.644} C_VEL
LIN {X 0,Y 594.39,Z 510.439,A -85,B 0,C 180,E1 -1024.578,E2 -1024.578} C_VEL
LIN {X 0,Y 594.385,Z 510.444,A -85,B 0,C 180,E1 -1027.086,E2 -1027.086} C_VEL
LIN {X 0,Y 594.374,Z 510.445,A -85,B 0,C 180,E1 -1029.774,E2 -1029.774} C_VEL
LIN {X 0,Y 594.37,Z 510.441,A -85,B 0,C 180,E1 -1032.374,E2 -1032.374} C_VEL
LIN {X 0,Y 594.359,Z 510.448,A -85,B 0,C 180,E1 -1035.19,E2 -1035.19} C_VEL
LIN {X 0,Y 594.379,Z 510.441,A -85,B 0,C 180,E1 -1038.151,E2 -1038.151} C_VEL
LIN {X 0,Y 594.391,Z 510.438,A -85,B 0,C 180,E1 -1040.321,E2 -1040.321} C_VEL
LIN {X 0,Y 594.38,Z 510.441,A -85,B 0,C 180,E1 -1042.913,E2 -1042.913} C_VEL
LIN {X 0,Y 594.383,Z 510.444,A -85,B 0,C 180,E1 -1045.86,E2 -1045.86} C_VEL
LIN {X 0,Y 594.385,Z 510.44,A -85,B 0,C 180,E1 -1048.65,E2 -1048.65} C_VEL
LIN {X 0,Y 594.383,Z 510.443,A -85,B 0,C 180,E1 -1051.04,E2 -1051.04} C_VEL
LIN {X 0,Y 594.39,Z 510.442,A -85,B 0,C 180,E1 -1053.974,E2 -1053.974} C_VEL
LIN {X 0,Y 594.387,Z 510.439,A -85,B 0,C 180,E1 -1056.296,E2 -1056.296} C_VEL
LIN {X 0,Y 594.404,Z 510.442,A -85,B 0,C 180,E1 -1059.224,E2 -1059.224} C_VEL
LIN {X 0,Y 594.374,Z 510.442,A -85,B 0,C 180,E1 -1062.096,E2 -1062.096} C_VEL
LIN {X 0,Y 594.364,Z 510.442,A -85,B 0,C 180,E1 -1064.219,E2 -1064.219} C_VEL
LIN {X 0,Y 594.365,Z 510.445,A -85,B 0,C 180,E1 -1067.017,E2 -1067.017} C_VEL
LIN {X 0,Y 594.391,Z 510.444,A -85,B 0,C 180,E1 -1069.784,E2 -1069.784} C_VEL
LIN {X 0,Y 594.387,Z 510.439,A -85,B 0,C 180,E1 -1072.527,E2 -1072.527} C_VEL
LIN {X 0,Y 594.396,Z 510.444,A -85,B 0,C 180,E1 -1075.252,E2 -1075.252} C_VEL
LIN {X 0,Y 594.391,Z 510.442,A -85,B 0,C 180,E1 -1077.967,E2 -1077.967} C_VEL
LIN {X 0,Y 594.42,Z 510.435,A -85,B 0,C 180,E1 -1080.677,E2 -1080.677} C_VEL
LIN {X 0,Y 594.378,Z 510.447,A -85,B 0,C 180,E1 -1083.389,E2 -1083.389} C_VEL
LIN {X 0,Y 594.364,Z 510.444,A -85,B 0,C 180,E1 -1086.109,E2 -1086.109} C_VEL
LIN {X 0,Y 594.395,Z 510.439,A -85,B 0,C 180,E1 -1088.842,E2 -1088.842} C_VEL
LIN {X 0,Y 594.387,Z 510.45,A -85,B 0,C 180,E1 -1091.596,E2 -1091.596} C_VEL
LIN {X 0,Y 594.383,Z 510.44,A -85,B 0,C 180,E1 -1094.377,E2 -1094.377} C_VEL
LIN {X 0,Y 594.384,Z 510.443,A -85,B 0,C 180,E1 -1097.194,E2 -1097.194} C_VEL
LIN {X 0,Y 594.371,Z 510.445,A -85,B 0,C 180,E1 -1100.054,E2 -1100.054} C_VEL
LIN {X 0,Y 594.358,Z 510.444,A -85,B 0,C 180,E1 -1102.968,E2 -1102.968} C_VEL
LIN {X 0,Y 594.374,Z 510.444,A -85,B 0,C 180,E1 -1105.193,E2 -1105.193} C_VEL
LIN {X 0,Y 594.378,Z 510.449,A -85,B 0,C 180,E1 -1107.527,E2 -1107.527} C_VEL
LIN {X 0,Y 594.381,Z 510.441,A -85,B 0,C 180,E1 -1110.329,E2 -1110.329} C_VEL
LIN {X 0,Y 594.373,Z 510.442,A -85,B 0,C 180,E1 -1112.951,E2 -1112.951} C_VEL
LIN {X 0,Y 594.381,Z 510.446,A -85,B 0,C 180,E1 -1115.407,E2 -1115.407} C_VEL
LIN {X 0,Y 594.38,Z 510.446,A -85,B 0,C 180,E1 -1117.941,E2 -1117.941} C_VEL
LIN {X 0,Y 594.373,Z 510.441,A -85,B 0,C 180,E1 -1120.823,E2 -1120.823} C_VEL
LIN {X 0,Y 594.362,Z 510.446,A -85,B 0,C 180,E1 -1123.3,E2 -1123.3} C_VEL
LIN {X 0,Y 594.379,Z 510.443,A -85,B 0,C 180,E1 -1126.16,E2 -1126.16} C_VEL
LIN {X 0,Y 594.38,Z 510.44,A -85,B 0,C 180,E1 -1128.537,E2 -1128.537} C_VEL
LIN {X 0,Y 594.386,Z 510.443,A -85,B 0,C 180,E1 -1131.296,E2 -1131.296} C_VEL
LIN {X 0,Y 594.393,Z 510.449,A -85,B 0,C 180,E1 -1133.759,E2 -1133.759} C_VEL
LIN {X 0,Y 594.377,Z 510.442,A -85,B 0,C 180,E1 -1136.24,E2 -1136.24} C_VEL
LIN {X 0,Y 594.39,Z 510.434,A -85,B 0,C 180,E1 -1138.652,E2 -1138.652} C_VEL
LIN {X 0,Y 594.381,Z 510.441,A -85,B 0,C 180,E1 -1141.043,E2 -1141.043} C_VEL
LIN {X 0,Y 594.382,Z 510.446,A -85,B 0,C 180,E1 -1143.979,E2 -1143.979} C_VEL
LIN {X 0,Y 594.391,Z 510.445,A -85,B 0,C 180,E1 -1146.297,E2 -1146.297} C_VEL
LIN {X 0,Y 594.411,Z 510.663,A -85,B 0,C 180,E1 -1147.412,E2 -1147.412} C_VEL
LIN {X 0,Y 594.741,Z 514.248,A -85,B 0,C 180,E1 -1147.965,E2 -1147.965} C_VEL
LIN {X 0,Y 594.633,Z 534.718,A -85,B 0,C 180,E1 -1150.9,E2 -1150.9} C_VEL
LIN {X 0,Y 594.512,Z 554.547,A -85,B 0,C 180,E1 -1153.695,E2 -1153.695} C_VEL
LIN {X 0,Y 594.428,Z 574.696,A -85,B 0,C 180,E1 -1156.497,E2 -1156.497} C_VEL
LIN {X 0,Y 594.445,Z 576.029,A -85,B 0,C 180,E1 -1156.65,E2 -1156.65} C_VEL
LIN {X 0,Y 594.78,Z 579.779,A -85,B 0,C 180,E1 -1156.723,E2 -1156.723} C_VEL
LIN {X 0,Y 594.663,Z 683.984,A -85,B 0,C 180,E1 -1158,E2 -1158} C_VEL
LIN {X 0,Y 594.637,Z 697.24,A -85,B 0,C 180,E1 -1158.302,E2 -1158.302} C_VEL
LIN {X 0,Y 594.594,Z 709.581,A -85,B 0,C 180,E1 -1158.719,E2 -1158.719} C_VEL
LIN {X 0,Y 594.539,Z 721.646,A -85,B 0,C 180,E1 -1159.271,E2 -1159.271} C_VEL
LIN {X 0,Y 594.468,Z 733.21,A -85,B 0,C 180,E1 -1159.958,E2 -1159.958} C_VEL
LIN {X 0,Y 594.413,Z 743.604,A -85,B 0,C 180,E1 -1160.73,E2 -1160.73} C_VEL
LIN {X 0,Y 594.383,Z 752.119,A -85,B 0,C 180,E1 -1161.501,E2 -1161.501} C_VEL
LIN {X 0,Y 594.347,Z 759.966,A -85,B 0,C 180,E1 -1162.356,E2 -1162.356} C_VEL
LIN {X 0,Y 594.282,Z 767.816,A -85,B 0,C 180,E1 -1163.409,E2 -1163.409} C_VEL
LIN {X 0,Y 594.289,Z 774.684,A -85,B 0,C 180,E1 -1164.572,E2 -1164.572} C_VEL
LIN {X 0,Y 594.27,Z 779.374,A -85,B 0,C 180,E1 -1165.592,E2 -1165.592} C_VEL
LIN {X 0,Y 594.268,Z 782.959,A -85,B 0,C 180,E1 -1166.611,E2 -1166.611} C_VEL
LIN {X 0,Y 594.226,Z 784.811,A -85,B 0,C 180,E1 -1167.289,E2 -1167.289} C_VEL
LIN {X 0,Y 594.239,Z 786.203,A -85,B 0,C 180,E1 -1167.967,E2 -1167.967} C_VEL
LIN {X 0,Y 594.239,Z 787.784,A -85,B 0,C 180,E1 -1169.323,E2 -1169.323} C_VEL
LIN {X 0,Y 594.236,Z 788,A -85,B 0,C 180,E1 -1170.001,E2 -1170.001} C_VEL
LIN {X 0,Y 594.247,Z 787.184,A -85,B 0,C 180,E1 -1171.356,E2 -1171.356} C_VEL
LIN {X 0,Y 594.239,Z 786.201,A -85,B 0,C 180,E1 -1172.034,E2 -1172.034} C_VEL
LIN {X 0,Y 594.226,Z 784.807,A -85,B 0,C 180,E1 -1172.712,E2 -1172.712} C_VEL
LIN {X 0,Y 594.288,Z 781.894,A -85,B 0,C 180,E1 -1173.73,E2 -1173.73} C_VEL
LIN {X 0,Y 594.242,Z 777.948,A -85,B 0,C 180,E1 -1174.749,E2 -1174.749} C_VEL
LIN {X 0,Y 594.304,Z 771.874,A -85,B 0,C 180,E1 -1175.94,E2 -1175.94} C_VEL
LIN {X 0,Y 594.309,Z 765.232,A -85,B 0,C 180,E1 -1176.963,E2 -1176.963} C_VEL
LIN {X 0,Y 594.359,Z 756.985,A -85,B 0,C 180,E1 -1177.987,E2 -1177.987} C_VEL
LIN {X 0,Y 594.382,Z 748.531,A -85,B 0,C 180,E1 -1178.843,E2 -1178.843} C_VEL
LIN {X 0,Y 594.424,Z 738.086,A -85,B 0,C 180,E1 -1179.7,E2 -1179.7} C_VEL
LIN {X 0,Y 594.49,Z 727.749,A -85,B 0,C 180,E1 -1180.387,E2 -1180.387} C_VEL
LIN {X 0,Y 594.561,Z 716.686,A -85,B 0,C 180,E1 -1180.975,E2 -1180.975} C_VEL
LIN {X 0,Y 594.601,Z 704.689,A -85,B 0,C 180,E1 -1181.465,E2 -1181.465} C_VEL
LIN {X 0,Y 594.648,Z 691.331,A -85,B 0,C 180,E1 -1181.851,E2 -1181.851} C_VEL
LIN {X 0,Y 594.697,Z 678.043,A -85,B 0,C 180,E1 -1182.088,E2 -1182.088} C_VEL
LIN {X 0,Y 594.623,Z 577.329,A -85,B 0,C 180,E1 -1183.311,E2 -1183.311} C_VEL
LIN {X 0,Y 594.44,Z 575.718,A -85,B 0,C 180,E1 -1183.373,E2 -1183.373} C_VEL
LIN {X 0,Y 594.513,Z 554.537,A -85,B 0,C 180,E1 -1186.306,E2 -1186.306} C_VEL
LIN {X 0,Y 594.635,Z 534.715,A -85,B 0,C 180,E1 -1189.1,E2 -1189.1} C_VEL
LIN {X 0,Y 594.742,Z 514.239,A -85,B 0,C 180,E1 -1192.036,E2 -1192.036} C_VEL
LIN {X 0,Y 594.414,Z 510.549,A -85,B 0,C 180,E1 -1192.624,E2 -1192.624} C_VEL
LIN {X 0,Y 594.376,Z 510.442,A -85,B 0,C 180,E1 -1195.194,E2 -1195.194} C_VEL
LIN {X 0,Y 594.391,Z 510.441,A -85,B 0,C 180,E1 -1197.527,E2 -1197.527} C_VEL
LIN {X 0,Y 594.39,Z 510.447,A -85,B 0,C 180,E1 -1200.328,E2 -1200.328} C_VEL
LIN {X 0,Y 594.38,Z 510.441,A -85,B 0,C 180,E1 -1202.95,E2 -1202.95} C_VEL
LIN {X 0,Y 594.352,Z 510.445,A -85,B 0,C 180,E1 -1205.409,E2 -1205.409} C_VEL
LIN {X 0,Y 594.391,Z 510.447,A -85,B 0,C 180,E1 -1207.941,E2 -1207.941} C_VEL
LIN {X 0,Y 594.38,Z 510.441,A -85,B 0,C 180,E1 -1210.822,E2 -1210.822} C_VEL
LIN {X 0,Y 594.388,Z 510.448,A -85,B 0,C 180,E1 -1213.841,E2 -1213.841} C_VEL
LIN {X 0,Y 594.37,Z 510.443,A -85,B 0,C 180,E1 -1216.701,E2 -1216.701} C_VEL
LIN {X 0,Y 594.375,Z 510.444,A -85,B 0,C 180,E1 -1219.433,E2 -1219.433} C_VEL
LIN {X 0,Y 594.392,Z 510.442,A -85,B 0,C 180,E1 -1222.392,E2 -1222.392} C_VEL
LIN {X 0,Y 594.388,Z 510.44,A -85,B 0,C 180,E1 -1224.672,E2 -1224.672} C_VEL
LIN {X 0,Y 594.383,Z 510.441,A -85,B 0,C 180,E1 -1227.088,E2 -1227.088} C_VEL
LIN {X 0,Y 594.389,Z 510.448,A -85,B 0,C 180,E1 -1229.672,E2 -1229.672} C_VEL
LIN {X 0,Y 594.378,Z 510.442,A -85,B 0,C 180,E1 -1232.539,E2 -1232.539} C_VEL
LIN {X 0,Y 594.418,Z 510.592,A -85,B 0,C 180,E1 -1235.26,E2 -1235.26} C_VEL
LIN {X 0,Y 594.926,Z 513.996,A -85,B 0,C 180,E1 -1235.763,E2 -1235.763} C_VEL
LIN {X 0,Y 594.788,Z 533.883,A -85,B 0,C 180,E1 -1238.331,E2 -1238.331} C_VEL
LIN {X 0,Y 594.688,Z 556.901,A -85,B 0,C 180,E1 -1241.25,E2 -1241.25} C_VEL
LIN {X 0,Y 594.554,Z 582.184,A -85,B 0,C 180,E1 -1244.4,E2 -1244.4} C_VEL
LIN {X 0,Y 594.459,Z 606.336,A -85,B 0,C 180,E1 -1247.366,E2 -1247.366} C_VEL
LIN {X 0,Y 594.386,Z 630.96,A -85,B 0,C 180,E1 -1250.343,E2 -1250.343} C_VEL
LIN {X 0,Y 594.513,Z 634.055,A -85,B 0,C 180,E1 -1250.409,E2 -1250.409} C_VEL
LIN {X 0,Y 594.492,Z 702.126,A -85,B 0,C 180,E1 -1251.245,E2 -1251.245} C_VEL
LIN {X 0,Y 594.456,Z 712.996,A -85,B 0,C 180,E1 -1251.502,E2 -1251.502} C_VEL
LIN {X 0,Y 594.441,Z 722.415,A -85,B 0,C 180,E1 -1251.844,E2 -1251.844} C_VEL
LIN {X 0,Y 594.413,Z 731.137,A -85,B 0,C 180,E1 -1252.271,E2 -1252.271} C_VEL
LIN {X 0,Y 594.361,Z 739.356,A -85,B 0,C 180,E1 -1252.783,E2 -1252.783} C_VEL
LIN {X 0,Y 594.344,Z 746.788,A -85,B 0,C 180,E1 -1253.357,E2 -1253.357} C_VEL
LIN {X 0,Y 594.326,Z 754.173,A -85,B 0,C 180,E1 -1254.061,E2 -1254.061} C_VEL
LIN {X 0,Y 594.262,Z 761.143,A -85,B 0,C 180,E1 -1254.911,E2 -1254.911} C_VEL
LIN {X 0,Y 594.284,Z 765.627,A -85,B 0,C 180,E1 -1255.591,E2 -1255.591} C_VEL
LIN {X 0,Y 594.268,Z 770.813,A -85,B 0,C 180,E1 -1256.61,E2 -1256.61} C_VEL
LIN {X 0,Y 594.235,Z 773.412,A -85,B 0,C 180,E1 -1257.288,E2 -1257.288} C_VEL
LIN {X 0,Y 594.235,Z 775.395,A -85,B 0,C 180,E1 -1257.967,E2 -1257.967} C_VEL
LIN {X 0,Y 594.243,Z 776.824,A -85,B 0,C 180,E1 -1258.645,E2 -1258.645} C_VEL
LIN {X 0,Y 594.234,Z 777.691,A -85,B 0,C 180,E1 -1259.322,E2 -1259.322} C_VEL
LIN {X 0,Y 594.234,Z 777.996,A -85,B 0,C 180,E1 -1260,E2 -1260} C_VEL
LIN {X 0,Y 594.237,Z 777.743,A -85,B 0,C 180,E1 -1260.678,E2 -1260.678} C_VEL
LIN {X 0,Y 594.247,Z 776.949,A -85,B 0,C 180,E1 -1261.355,E2 -1261.355} C_VEL
LIN {X 0,Y 594.235,Z 775.607,A -85,B 0,C 180,E1 -1262.033,E2 -1262.033} C_VEL
LIN {X 0,Y 594.25,Z 772.571,A -85,B 0,C 180,E1 -1263.051,E2 -1263.051} C_VEL
LIN {X 0,Y 594.262,Z 768.042,A -85,B 0,C 180,E1 -1264.069,E2 -1264.069} C_VEL
LIN {X 0,Y 594.307,Z 762.944,A -85,B 0,C 180,E1 -1264.918,E2 -1264.918} C_VEL
LIN {X 0,Y 594.32,Z 756.456,A -85,B 0,C 180,E1 -1265.769,E2 -1265.769} C_VEL
LIN {X 0,Y 594.337,Z 747.925,A -85,B 0,C 180,E1 -1266.637,E2 -1266.637} C_VEL
LIN {X 0,Y 594.36,Z 739.421,A -85,B 0,C 180,E1 -1267.303,E2 -1267.303} C_VEL
LIN {X 0,Y 594.402,Z 731.215,A -85,B 0,C 180,E1 -1267.815,E2 -1267.815} C_VEL
LIN {X 0,Y 594.442,Z 720.46,A -85,B 0,C 180,E1 -1268.327,E2 -1268.327} C_VEL
LIN {X 0,Y 594.442,Z 709.977,A -85,B 0,C 180,E1 -1268.67,E2 -1268.67} C_VEL
LIN {X 0,Y 594.455,Z 699.786,A -85,B 0,C 180,E1 -1268.884,E2 -1268.884} C_VEL
LIN {X 0,Y 594.524,Z 659.837,A -85,B 0,C 180,E1 -1269.371,E2 -1269.371} C_VEL
LIN {X 0,Y 593.892,Z 655.953,A -85,B 0,C 180,E1 -1269.428,E2 -1269.428} C_VEL
LIN {X 0,Y 588.217,Z 643.935,A -85,B 0,C 180,E1 -1269.665,E2 -1269.665} C_VEL
LIN {X 0,Y 587.531,Z 640.05,A -85,B 0,C 180,E1 -1269.723,E2 -1269.723} C_VEL
LIN {X 0,Y 587.35,Z 631.435,A -85,B 0,C 180,E1 -1269.839,E2 -1269.839} C_VEL
LIN {X 0,Y 587.329,Z 629.807,A -85,B 0,C 180,E1 -1269.992,E2 -1269.992} C_VEL
LIN {X 0,Y 587.439,Z 605.646,A -85,B 0,C 180,E1 -1272.963,E2 -1272.963} C_VEL
LIN {X 0,Y 587.565,Z 582.906,A -85,B 0,C 180,E1 -1275.79,E2 -1275.79} C_VEL
LIN {X 0,Y 587.702,Z 560.165,A -85,B 0,C 180,E1 -1278.656,E2 -1278.656} C_VEL
LIN {X 0,Y 587.863,Z 537.492,A -85,B 0,C 180,E1 -1281.56,E2 -1281.56} C_VEL
LIN {X 0,Y 588.056,Z 517.588,A -85,B 0,C 180,E1 -1284.154,E2 -1284.154} C_VEL
LIN {X 0,Y 587.758,Z 513.258,A -85,B 0,C 180,E1 -1284.74,E2 -1284.74} C_VEL
LIN {X 0,Y 587.353,Z 511.372,A -85,B 0,C 180,E1 -1285.066,E2 -1285.066} C_VEL
LIN {X 0,Y 587.345,Z 511.32,A -85,B 0,C 180,E1 -1287.818,E2 -1287.818} C_VEL
LIN {X 0,Y 587.339,Z 511.327,A -85,B 0,C 180,E1 -1290.51,E2 -1290.51} C_VEL
LIN {X 0,Y 587.338,Z 511.318,A -85,B 0,C 180,E1 -1293.397,E2 -1293.397} C_VEL
LIN {X 0,Y 587.36,Z 511.317,A -85,B 0,C 180,E1 -1295.895,E2 -1295.895} C_VEL
LIN {X 0,Y 587.335,Z 511.329,A -85,B 0,C 180,E1 -1298.479,E2 -1298.479} C_VEL
LIN {X 0,Y 587.338,Z 511.316,A -85,B 0,C 180,E1 -1301.157,E2 -1301.157} C_VEL
LIN {X 0,Y 587.331,Z 511.319,A -85,B 0,C 180,E1 -1304.113,E2 -1304.113} C_VEL
LIN {X 0,Y 587.326,Z 511.322,A -85,B 0,C 180,E1 -1306.994,E2 -1306.994} C_VEL
LIN {X 0,Y 587.321,Z 511.318,A -85,B 0,C 180,E1 -1309.746,E2 -1309.746} C_VEL
LIN {X 0,Y 587.35,Z 511.322,A -85,B 0,C 180,E1 -1312.392,E2 -1312.392} C_VEL
LIN {X 0,Y 587.363,Z 511.314,A -85,B 0,C 180,E1 -1315.78,E2 -1315.78} C_VEL
LIN {X 0,Y 587.35,Z 511.32,A -85,B 0,C 180,E1 -1318.231,E2 -1318.231} C_VEL
LIN {X 0,Y 587.354,Z 511.322,A -85,B 0,C 180,E1 -1320.867,E2 -1320.867} C_VEL
LIN {X 0,Y 587.362,Z 511.315,A -85,B 0,C 180,E1 -1323.819,E2 -1323.819} C_VEL
LIN {X 0,Y 587.341,Z 511.317,A -85,B 0,C 180,E1 -1325.993,E2 -1325.993} C_VEL
LIN {X 0,Y 587.325,Z 511.323,A -85,B 0,C 180,E1 -1328.225,E2 -1328.225} C_VEL
LIN {X 0,Y 587.399,Z 511.5,A -85,B 0,C 180,E1 -1330.463,E2 -1330.463} C_VEL
LIN {X 0,Y 587.496,Z 520.641,A -85,B 0,C 180,E1 -1332.058,E2 -1332.058} C_VEL
LIN {X 0,Y 587.41,Z 537.413,A -85,B 0,C 180,E1 -1334.916,E2 -1334.916} C_VEL
LIN {X 0,Y 587.397,Z 547.163,A -85,B 0,C 180,E1 -1336.529,E2 -1336.529} C_VEL
LIN {X 0,Y 587.75,Z 549.596,A -85,B 0,C 180,E1 -1336.604,E2 -1336.604} C_VEL
LIN {X 0,Y 587.743,Z 653.854,A -85,B 0,C 180,E1 -1337.899,E2 -1337.899} C_VEL
LIN {X 0,Y 587.705,Z 667.159,A -85,B 0,C 180,E1 -1338.204,E2 -1338.204} C_VEL
LIN {X 0,Y 587.615,Z 679.731,A -85,B 0,C 180,E1 -1338.634,E2 -1338.634} C_VEL
LIN {X 0,Y 587.56,Z 690.764,A -85,B 0,C 180,E1 -1339.141,E2 -1339.141} C_VEL
LIN {X 0,Y 587.475,Z 702.532,A -85,B 0,C 180,E1 -1339.836,E2 -1339.836} C_VEL
LIN {X 0,Y 587.393,Z 713.042,A -85,B 0,C 180,E1 -1340.617,E2 -1340.617} C_VEL
LIN {X 0,Y 587.323,Z 721.646,A -85,B 0,C 180,E1 -1341.397,E2 -1341.397} C_VEL
LIN {X 0,Y 587.274,Z 729.573,A -85,B 0,C 180,E1 -1342.262,E2 -1342.262} C_VEL
LIN {X 0,Y 587.234,Z 736.145,A -85,B 0,C 180,E1 -1343.126,E2 -1343.126} C_VEL
LIN {X 0,Y 587.237,Z 742.615,A -85,B 0,C 180,E1 -1344.161,E2 -1344.161} C_VEL
LIN {X 0,Y 587.146,Z 747.756,A -85,B 0,C 180,E1 -1345.193,E2 -1345.193} C_VEL
LIN {X 0,Y 587.213,Z 751.745,A -85,B 0,C 180,E1 -1346.225,E2 -1346.225} C_VEL
LIN {X 0,Y 587.131,Z 754.695,A -85,B 0,C 180,E1 -1347.255,E2 -1347.255} C_VEL
LIN {X 0,Y 587.14,Z 756.127,A -85,B 0,C 180,E1 -1347.941,E2 -1347.941} C_VEL
LIN {X 0,Y 587.14,Z 757.753,A -85,B 0,C 180,E1 -1349.314,E2 -1349.314} C_VEL
LIN {X 0,Y 587.137,Z 757.996,A -85,B 0,C 180,E1 -1349.999,E2 -1349.999} C_VEL
LIN {X 0,Y 587.14,Z 757.815,A -85,B 0,C 180,E1 -1350.685,E2 -1350.685} C_VEL
LIN {X 0,Y 587.14,Z 756.276,A -85,B 0,C 180,E1 -1352.057,E2 -1352.057} C_VEL
LIN {X 0,Y 587.132,Z 754.915,A -85,B 0,C 180,E1 -1352.744,E2 -1352.744} C_VEL
LIN {X 0,Y 587.213,Z 752.038,A -85,B 0,C 180,E1 -1353.774,E2 -1353.774} C_VEL
LIN {X 0,Y 587.147,Z 748.139,A -85,B 0,C 180,E1 -1354.806,E2 -1354.806} C_VEL
LIN {X 0,Y 587.229,Z 743.108,A -85,B 0,C 180,E1 -1355.838,E2 -1355.838} C_VEL
LIN {X 0,Y 587.23,Z 736.788,A -85,B 0,C 180,E1 -1356.873,E2 -1356.873} C_VEL
LIN {X 0,Y 587.288,Z 728.87,A -85,B 0,C 180,E1 -1357.909,E2 -1357.909} C_VEL
LIN {X 0,Y 587.343,Z 719.024,A -85,B 0,C 180,E1 -1358.948,E2 -1358.948} C_VEL
LIN {X 0,Y 587.418,Z 708.706,A -85,B 0,C 180,E1 -1359.816,E2 -1359.816} C_VEL
LIN {X 0,Y 587.493,Z 698.502,A -85,B 0,C 180,E1 -1360.511,E2 -1360.511} C_VEL
LIN {X 0,Y 587.578,Z 687.487,A -85,B 0,C 180,E1 -1361.112,E2 -1361.112} C_VEL
LIN {X 0,Y 587.638,Z 675.835,A -85,B 0,C 180,E1 -1361.607,E2 -1361.607} C_VEL
LIN {X 0,Y 587.716,Z 663.267,A -85,B 0,C 180,E1 -1361.991,E2 -1361.991} C_VEL
LIN {X 0,Y 587.791,Z 649.733,A -85,B 0,C 180,E1 -1362.252,E2 -1362.252} C_VEL
LIN {X 0,Y 587.775,Z 549.858,A -85,B 0,C 180,E1 -1363.482,E2 -1363.482} C_VEL
LIN {X 0,Y 587.409,Z 547.204,A -85,B 0,C 180,E1 -1363.557,E2 -1363.557} C_VEL
LIN {X 0,Y 587.44,Z 530.611,A -85,B 0,C 180,E1 -1366.328,E2 -1366.328} C_VEL
LIN {X 0,Y 587.548,Z 514.451,A -85,B 0,C 180,E1 -1369.097,E2 -1369.097} C_VEL
LIN {X 0,Y 587.393,Z 511.401,A -85,B 0,C 180,E1 -1369.663,E2 -1369.663} C_VEL
LIN {X 0,Y 587.32,Z 511.323,A -85,B 0,C 180,E1 -1372.868,E2 -1372.868} C_VEL
LIN {X 0,Y 587.336,Z 511.326,A -85,B 0,C 180,E1 -1375.516,E2 -1375.516} C_VEL
LIN {X 0,Y 587.348,Z 511.32,A -85,B 0,C 180,E1 -1377.817,E2 -1377.817} C_VEL
LIN {X 0,Y 587.342,Z 511.317,A -85,B 0,C 180,E1 -1380.51,E2 -1380.51} C_VEL
LIN {X 0,Y 587.339,Z 511.323,A -85,B 0,C 180,E1 -1383.111,E2 -1383.111} C_VEL
LIN {X 0,Y 587.354,Z 511.318,A -85,B 0,C 180,E1 -1385.895,E2 -1385.895} C_VEL
LIN {X 0,Y 587.332,Z 511.318,A -85,B 0,C 180,E1 -1388.478,E2 -1388.478} C_VEL
LIN {X 0,Y 587.336,Z 511.323,A -85,B 0,C 180,E1 -1391.156,E2 -1391.156} C_VEL
LIN {X 0,Y 587.331,Z 511.318,A -85,B 0,C 180,E1 -1394.113,E2 -1394.113} C_VEL
LIN {X 0,Y 587.311,Z 511.324,A -85,B 0,C 180,E1 -1396.993,E2 -1396.993} C_VEL
LIN {X 0,Y 587.325,Z 511.323,A -85,B 0,C 180,E1 -1399.746,E2 -1399.746} C_VEL
LIN {X 0,Y 587.34,Z 511.316,A -85,B 0,C 180,E1 -1402.392,E2 -1402.392} C_VEL
LIN {X 0,Y 587.347,Z 511.319,A -85,B 0,C 180,E1 -1404.946,E2 -1404.946} C_VEL
LIN {X 0,Y 587.338,Z 511.327,A -85,B 0,C 180,E1 -1407.421,E2 -1407.421} C_VEL
LIN {X 0,Y 587.342,Z 511.322,A -85,B 0,C 180,E1 -1409.83,E2 -1409.83} C_VEL
LIN {X 0,Y 587.346,Z 511.316,A -85,B 0,C 180,E1 -1412.306,E2 -1412.306} C_VEL
LIN {X 0,Y 587.336,Z 511.318,A -85,B 0,C 180,E1 -1414.483,E2 -1414.483} C_VEL
LIN {X 0,Y 587.336,Z 511.328,A -85,B 0,C 180,E1 -1417.486,E2 -1417.486} C_VEL
LIN {X 0,Y 587.329,Z 511.326,A -85,B 0,C 180,E1 -1419.695,E2 -1419.695} C_VEL
LIN {X 0,Y 587.352,Z 511.315,A -85,B 0,C 180,E1 -1422.594,E2 -1422.594} C_VEL
LIN {X 0,Y 587.358,Z 511.322,A -85,B 0,C 180,E1 -1425.739,E2 -1425.739} C_VEL
LIN {X 0,Y 587.336,Z 511.318,A -85,B 0,C 180,E1 -1428.263,E2 -1428.263} C_VEL
LIN {X 0,Y 587.34,Z 511.319,A -85,B 0,C 180,E1 -1431.051,E2 -1431.051} C_VEL
LIN {X 0,Y 587.368,Z 511.319,A -85,B 0,C 180,E1 -1433.264,E2 -1433.264} C_VEL
LIN {X 0,Y 587.312,Z 511.324,A -85,B 0,C 180,E1 -1435.883,E2 -1435.883} C_VEL
LIN {X 0,Y 587.361,Z 511.318,A -85,B 0,C 180,E1 -1437.943,E2 -1437.943} C_VEL
LIN {X 0,Y 587.39,Z 511.311,A -85,B 0,C 180,E1 -1440.686,E2 -1440.686} C_VEL
LIN {X 0,Y 587.33,Z 511.326,A -85,B 0,C 180,E1 -1443.43,E2 -1443.43} C_VEL
LIN {X 0,Y 587.35,Z 511.325,A -85,B 0,C 180,E1 -1445.493,E2 -1445.493} C_VEL
LIN {X 0,Y 587.366,Z 511.315,A -85,B 0,C 180,E1 -1448.255,E2 -1448.255} C_VEL
LIN {X 0,Y 587.34,Z 511.32,A -85,B 0,C 180,E1 -1451.134,E2 -1451.134} C_VEL
LIN {X 0,Y 587.352,Z 511.322,A -85,B 0,C 180,E1 -1453.846,E2 -1453.846} C_VEL
LIN {X 0,Y 587.355,Z 511.315,A -85,B 0,C 180,E1 -1456.819,E2 -1456.819} C_VEL
LIN {X 0,Y 587.338,Z 511.328,A -85,B 0,C 180,E1 -1459.575,E2 -1459.575} C_VEL
LIN {X 0,Y 587.317,Z 511.327,A -85,B 0,C 180,E1 -1461.775,E2 -1461.775} C_VEL
LIN {X 0,Y 587.346,Z 511.317,A -85,B 0,C 180,E1 -1464.759,E2 -1464.759} C_VEL
LIN {X 0,Y 587.324,Z 511.32,A -85,B 0,C 180,E1 -1467.047,E2 -1467.047} C_VEL
LIN {X 0,Y 587.343,Z 511.323,A -85,B 0,C 180,E1 -1469.38,E2 -1469.38} C_VEL
LIN {X 0,Y 587.35,Z 511.323,A -85,B 0,C 180,E1 -1471.838,E2 -1471.838} C_VEL
LIN {X 0,Y 587.352,Z 511.316,A -85,B 0,C 180,E1 -1474.35,E2 -1474.35} C_VEL
LIN {X 0,Y 587.348,Z 511.314,A -85,B 0,C 180,E1 -1476.747,E2 -1476.747} C_VEL
LIN {X 0,Y 587.342,Z 511.322,A -85,B 0,C 180,E1 -1479.36,E2 -1479.36} C_VEL
LIN {X 0,Y 587.33,Z 511.321,A -85,B 0,C 180,E1 -1482.108,E2 -1482.108} C_VEL
LIN {X 0,Y 587.312,Z 511.323,A -85,B 0,C 180,E1 -1485.09,E2 -1485.09} C_VEL
LIN {X 0,Y 587.349,Z 511.323,A -85,B 0,C 180,E1 -1487.928,E2 -1487.928} C_VEL
LIN {X 0,Y 587.332,Z 511.319,A -85,B 0,C 180,E1 -1491.059,E2 -1491.059} C_VEL
LIN {X 0,Y 587.352,Z 511.318,A -85,B 0,C 180,E1 -1493.292,E2 -1493.292} C_VEL
LIN {X 0,Y 587.36,Z 511.323,A -85,B 0,C 180,E1 -1495.781,E2 -1495.781} C_VEL
LIN {X 0,Y 587.352,Z 511.311,A -85,B 0,C 180,E1 -1498.233,E2 -1498.233} C_VEL
LIN {X 0,Y 587.348,Z 511.316,A -85,B 0,C 180,E1 -1500.867,E2 -1500.867} C_VEL
LIN {X 0,Y 587.358,Z 511.32,A -85,B 0,C 180,E1 -1503.82,E2 -1503.82} C_VEL
LIN {X 0,Y 587.338,Z 511.326,A -85,B 0,C 180,E1 -1505.994,E2 -1505.994} C_VEL
LIN {X 0,Y 587.352,Z 511.402,A -85,B 0,C 180,E1 -1507.21,E2 -1507.21} C_VEL
LIN {X 0,Y 587.833,Z 515.508,A -85,B 0,C 180,E1 -1507.877,E2 -1507.877} C_VEL
LIN {X 0,Y 587.675,Z 536.122,A -85,B 0,C 180,E1 -1510.867,E2 -1510.867} C_VEL
LIN {X 0,Y 587.517,Z 555.806,A -85,B 0,C 180,E1 -1513.674,E2 -1513.674} C_VEL
LIN {X 0,Y 587.41,Z 575.531,A -85,B 0,C 180,E1 -1516.443,E2 -1516.443} C_VEL
LIN {X 0,Y 587.557,Z 576.981,A -85,B 0,C 180,E1 -1516.521,E2 -1516.521} C_VEL
LIN {X 0,Y 587.861,Z 583.356,A -85,B 0,C 180,E1 -1516.608,E2 -1516.608} C_VEL
LIN {X 0,Y 587.724,Z 683.983,A -85,B 0,C 180,E1 -1517.856,E2 -1517.856} C_VEL
LIN {X 0,Y 587.681,Z 697.239,A -85,B 0,C 180,E1 -1518.161,E2 -1518.161} C_VEL
LIN {X 0,Y 587.626,Z 709.763,A -85,B 0,C 180,E1 -1518.591,E2 -1518.591} C_VEL
LIN {X 0,Y 587.554,Z 721.645,A -85,B 0,C 180,E1 -1519.142,E2 -1519.142} C_VEL
LIN {X 0,Y 587.465,Z 733.211,A -85,B 0,C 180,E1 -1519.837,E2 -1519.837} C_VEL
LIN {X 0,Y 587.391,Z 743.605,A -85,B 0,C 180,E1 -1520.618,E2 -1520.618} C_VEL
LIN {X 0,Y 587.321,Z 752.119,A -85,B 0,C 180,E1 -1521.398,E2 -1521.398} C_VEL
LIN {X 0,Y 587.273,Z 759.966,A -85,B 0,C 180,E1 -1522.263,E2 -1522.263} C_VEL
LIN {X 0,Y 587.23,Z 766.475,A -85,B 0,C 180,E1 -1523.127,E2 -1523.127} C_VEL
LIN {X 0,Y 587.236,Z 772.87,A -85,B 0,C 180,E1 -1524.162,E2 -1524.162} C_VEL
LIN {X 0,Y 587.147,Z 777.952,A -85,B 0,C 180,E1 -1525.194,E2 -1525.194} C_VEL
LIN {X 0,Y 587.212,Z 781.898,A -85,B 0,C 180,E1 -1526.226,E2 -1526.226} C_VEL
LIN {X 0,Y 587.132,Z 784.811,A -85,B 0,C 180,E1 -1527.256,E2 -1527.256} C_VEL
LIN {X 0,Y 587.138,Z 786.202,A -85,B 0,C 180,E1 -1527.943,E2 -1527.943} C_VEL
LIN {X 0,Y 587.14,Z 787.785,A -85,B 0,C 180,E1 -1529.315,E2 -1529.315} C_VEL
LIN {X 0,Y 587.137,Z 788,A -85,B 0,C 180,E1 -1530.001,E2 -1530.001} C_VEL
LIN {X 0,Y 587.147,Z 787.184,A -85,B 0,C 180,E1 -1531.372,E2 -1531.372} C_VEL
LIN {X 0,Y 587.138,Z 786.2,A -85,B 0,C 180,E1 -1532.059,E2 -1532.059} C_VEL
LIN {X 0,Y 587.132,Z 784.807,A -85,B 0,C 180,E1 -1532.745,E2 -1532.745} C_VEL
LIN {X 0,Y 587.212,Z 781.894,A -85,B 0,C 180,E1 -1533.775,E2 -1533.775} C_VEL
LIN {X 0,Y 587.147,Z 777.948,A -85,B 0,C 180,E1 -1534.807,E2 -1534.807} C_VEL
LIN {X 0,Y 587.217,Z 771.874,A -85,B 0,C 180,E1 -1536.012,E2 -1536.012} C_VEL
LIN {X 0,Y 587.246,Z 765.232,A -85,B 0,C 180,E1 -1537.047,E2 -1537.047} C_VEL
LIN {X 0,Y 587.3,Z 756.985,A -85,B 0,C 180,E1 -1538.084,E2 -1538.084} C_VEL
LIN {X 0,Y 587.344,Z 748.531,A -85,B 0,C 180,E1 -1538.95,E2 -1538.95} C_VEL
LIN {X 0,Y 587.411,Z 738.087,A -85,B 0,C 180,E1 -1539.817,E2 -1539.817} C_VEL
LIN {X 0,Y 587.492,Z 727.749,A -85,B 0,C 180,E1 -1540.512,E2 -1540.512} C_VEL
LIN {X 0,Y 587.585,Z 715.791,A -85,B 0,C 180,E1 -1541.149,E2 -1541.149} C_VEL
LIN {X 0,Y 587.64,Z 703.579,A -85,B 0,C 180,E1 -1541.64,E2 -1541.64} C_VEL
LIN {X 0,Y 587.729,Z 690.416,A -85,B 0,C 180,E1 -1542.014,E2 -1542.014} C_VEL
LIN {X 0,Y 587.766,Z 678.043,A -85,B 0,C 180,E1 -1542.232,E2 -1542.232} C_VEL
LIN {X 0,Y 587.706,Z 577.885,A -85,B 0,C 180,E1 -1543.463,E2 -1543.463} C_VEL
LIN {X 0,Y 587.397,Z 575.716,A -85,B 0,C 180,E1 -1543.537,E2 -1543.537} C_VEL
LIN {X 0,Y 587.518,Z 555.797,A -85,B 0,C 180,E1 -1546.327,E2 -1546.327} C_VEL
LIN {X 0,Y 587.676,Z 536.12,A -85,B 0,C 180,E1 -1549.133,E2 -1549.133} C_VEL
LIN {X 0,Y 587.822,Z 515.499,A -85,B 0,C 180,E1 -1552.125,E2 -1552.125} C_VEL
LIN {X 0,Y 587.354,Z 511.407,A -85,B 0,C 180,E1 -1552.791,E2 -1552.791} C_VEL
LIN {X 0,Y 587.333,Z 511.32,A -85,B 0,C 180,E1 -1555.517,E2 -1555.517} C_VEL
LIN {X 0,Y 587.351,Z 511.321,A -85,B 0,C 180,E1 -1557.818,E2 -1557.818} C_VEL
LIN {X 0,Y 587.341,Z 511.322,A -85,B 0,C 180,E1 -1560.51,E2 -1560.51} C_VEL
LIN {X 0,Y 587.337,Z 511.319,A -85,B 0,C 180,E1 -1563.397,E2 -1563.397} C_VEL
LIN {X 0,Y 587.294,Z 511.331,A -85,B 0,C 180,E1 -1565.9,E2 -1565.9} C_VEL
LIN {X 0,Y 587.333,Z 511.322,A -85,B 0,C 180,E1 -1568.48,E2 -1568.48} C_VEL
LIN {X 0,Y 587.34,Z 511.318,A -85,B 0,C 180,E1 -1571.157,E2 -1571.157} C_VEL
LIN {X 0,Y 587.339,Z 511.326,A -85,B 0,C 180,E1 -1574.114,E2 -1574.114} C_VEL
LIN {X 0,Y 587.317,Z 511.321,A -85,B 0,C 180,E1 -1576.994,E2 -1576.994} C_VEL
LIN {X 0,Y 587.323,Z 511.327,A -85,B 0,C 180,E1 -1579.746,E2 -1579.746} C_VEL
LIN {X 0,Y 587.347,Z 511.32,A -85,B 0,C 180,E1 -1582.392,E2 -1582.392} C_VEL
LIN {X 0,Y 587.353,Z 511.316,A -85,B 0,C 180,E1 -1584.946,E2 -1584.946} C_VEL
LIN {X 0,Y 587.343,Z 511.322,A -85,B 0,C 180,E1 -1587.421,E2 -1587.421} C_VEL
LIN {X 0,Y 587.337,Z 511.328,A -85,B 0,C 180,E1 -1589.83,E2 -1589.83} C_VEL
LIN {X 0,Y 587.345,Z 511.321,A -85,B 0,C 180,E1 -1592.309,E2 -1592.309} C_VEL
LIN {X 0,Y 587.348,Z 511.46,A -85,B 0,C 180,E1 -1595.052,E2 -1595.052} C_VEL
LIN {X 0,Y 588.078,Z 515.646,A -85,B 0,C 180,E1 -1595.68,E2 -1595.68} C_VEL
LIN {X 0,Y 587.901,Z 535.308,A -85,B 0,C 180,E1 -1598.248,E2 -1598.248} C_VEL
LIN {X 0,Y 587.735,Z 558.037,A -85,B 0,C 180,E1 -1601.164,E2 -1601.164} C_VEL
LIN {X 0,Y 587.565,Z 582.188,A -85,B 0,C 180,E1 -1604.21,E2 -1604.21} C_VEL
LIN {X 0,Y 587.442,Z 604.919,A -85,B 0,C 180,E1 -1607.037,E2 -1607.037} C_VEL
LIN {X 0,Y 587.332,Z 629.072,A -85,B 0,C 180,E1 -1610.008,E2 -1610.008} C_VEL
LIN {X 0,Y 587.356,Z 631.35,A -85,B 0,C 180,E1 -1610.248,E2 -1610.248} C_VEL
LIN {X 0,Y 587.519,Z 666.293,A -85,B 0,C 180,E1 -1610.685,E2 -1610.685} C_VEL
LIN {X 0,Y 587.49,Z 702.193,A -85,B 0,C 180,E1 -1611.14,E2 -1611.14} C_VEL
LIN {X 0,Y 587.45,Z 713.006,A -85,B 0,C 180,E1 -1611.399,E2 -1611.399} C_VEL
LIN {X 0,Y 587.424,Z 722.426,A -85,B 0,C 180,E1 -1611.746,E2 -1611.746} C_VEL
LIN {X 0,Y 587.373,Z 731.156,A -85,B 0,C 180,E1 -1612.178,E2 -1612.178} C_VEL
LIN {X 0,Y 587.303,Z 739.372,A -85,B 0,C 180,E1 -1612.695,E2 -1612.695} C_VEL
LIN {X 0,Y 587.298,Z 747.455,A -85,B 0,C 180,E1 -1613.333,E2 -1613.333} C_VEL
LIN {X 0,Y 587.254,Z 755.711,A -85,B 0,C 180,E1 -1614.162,E2 -1614.162} C_VEL
LIN {X 0,Y 587.232,Z 762.329,A -85,B 0,C 180,E1 -1615.022,E2 -1615.022} C_VEL
LIN {X 0,Y 587.184,Z 767.551,A -85,B 0,C 180,E1 -1615.882,E2 -1615.882} C_VEL
LIN {X 0,Y 587.18,Z 772.245,A -85,B 0,C 180,E1 -1616.913,E2 -1616.913} C_VEL
LIN {X 0,Y 587.135,Z 775.399,A -85,B 0,C 180,E1 -1617.942,E2 -1617.942} C_VEL
LIN {X 0,Y 587.142,Z 776.83,A -85,B 0,C 180,E1 -1618.628,E2 -1618.628} C_VEL
LIN {X 0,Y 587.135,Z 777.691,A -85,B 0,C 180,E1 -1619.314,E2 -1619.314} C_VEL
LIN {X 0,Y 587.135,Z 777.996,A -85,B 0,C 180,E1 -1620,E2 -1620} C_VEL
LIN {X 0,Y 587.137,Z 777.747,A -85,B 0,C 180,E1 -1620.686,E2 -1620.686} C_VEL
LIN {X 0,Y 587.147,Z 776.953,A -85,B 0,C 180,E1 -1621.372,E2 -1621.372} C_VEL
LIN {X 0,Y 587.134,Z 775.609,A -85,B 0,C 180,E1 -1622.058,E2 -1622.058} C_VEL
LIN {X 0,Y 587.159,Z 772.574,A -85,B 0,C 180,E1 -1623.088,E2 -1623.088} C_VEL
LIN {X 0,Y 587.184,Z 768.039,A -85,B 0,C 180,E1 -1624.118,E2 -1624.118} C_VEL
LIN {X 0,Y 587.214,Z 762.945,A -85,B 0,C 180,E1 -1624.978,E2 -1624.978} C_VEL
LIN {X 0,Y 587.255,Z 756.458,A -85,B 0,C 180,E1 -1625.839,E2 -1625.839} C_VEL
LIN {X 0,Y 587.269,Z 748.752,A -85,B 0,C 180,E1 -1626.643,E2 -1626.643} C_VEL
LIN {X 0,Y 587.312,Z 740.639,A -85,B 0,C 180,E1 -1627.305,E2 -1627.305} C_VEL
LIN {X 0,Y 587.373,Z 732.702,A -85,B 0,C 180,E1 -1627.823,E2 -1627.823} C_VEL
LIN {X 0,Y 587.393,Z 724.378,A -85,B 0,C 180,E1 -1628.255,E2 -1628.255} C_VEL
LIN {X 0,Y 587.435,Z 714.47,A -85,B 0,C 180,E1 -1628.644,E2 -1628.644} C_VEL
LIN {X 0,Y 587.498,Z 703.628,A -85,B 0,C 180,E1 -1628.925,E2 -1628.925} C_VEL
LIN {X 0,Y 587.504,Z 682.649,A -85,B 0,C 180,E1 -1629.207,E2 -1629.207} C_VEL
LIN {X 0,Y 587.531,Z 640.05,A -85,B 0,C 180,E1 -1629.723,E2 -1629.723} C_VEL
LIN {X 0,Y 587.181,Z 636.334,A -85,B 0,C 180,E1 -1629.816,E2 -1629.816} C_VEL
LIN {X 0,Y 585.783,Z 631.36,A -85,B 0,C 180,E1 -1630.082,E2 -1630.082} C_VEL
LIN {X 0,Y 583.918,Z 627.135,A -85,B 0,C 180,E1 -1630.447,E2 -1630.447} C_VEL
LIN {X 0,Y 581.474,Z 622.109,A -85,B 0,C 180,E1 -1631.047,E2 -1631.047} C_VEL
LIN {X 0,Y 580.435,Z 618.405,A -85,B 0,C 180,E1 -1631.528,E2 -1631.528} C_VEL
LIN {X 0,Y 580.35,Z 617.125,A -85,B 0,C 180,E1 -1631.689,E2 -1631.689} C_VEL
LIN {X 0,Y 580.467,Z 594.726,A -85,B 0,C 180,E1 -1634.493,E2 -1634.493} C_VEL
LIN {X 0,Y 580.666,Z 573.237,A -85,B 0,C 180,E1 -1637.213,E2 -1637.213} C_VEL
LIN {X 0,Y 580.849,Z 551.632,A -85,B 0,C 180,E1 -1639.987,E2 -1639.987} C_VEL
LIN {X 0,Y 581.116,Z 529.132,A -85,B 0,C 180,E1 -1642.924,E2 -1642.924} C_VEL
LIN {X 0,Y 581.222,Z 516.8,A -85,B 0,C 180,E1 -1644.562,E2 -1644.562} C_VEL
LIN {X 0,Y 580.335,Z 512.31,A -85,B 0,C 180,E1 -1645.246,E2 -1645.246} C_VEL
LIN {X 0,Y 580.301,Z 512.203,A -85,B 0,C 180,E1 -1648.186,E2 -1648.186} C_VEL
LIN {X 0,Y 580.287,Z 512.202,A -85,B 0,C 180,E1 -1650.694,E2 -1650.694} C_VEL
LIN {X 0,Y 580.307,Z 512.194,A -85,B 0,C 180,E1 -1653.316,E2 -1653.316} C_VEL
LIN {X 0,Y 580.33,Z 512.192,A -85,B 0,C 180,E1 -1655.767,E2 -1655.767} C_VEL
LIN {X 0,Y 580.292,Z 512.2,A -85,B 0,C 180,E1 -1658.146,E2 -1658.146} C_VEL
LIN {X 0,Y 580.302,Z 512.196,A -85,B 0,C 180,E1 -1660.843,E2 -1660.843} C_VEL
LIN {X 0,Y 580.282,Z 512.193,A -85,B 0,C 180,E1 -1663.658,E2 -1663.658} C_VEL
LIN {X 0,Y 580.29,Z 512.205,A -85,B 0,C 180,E1 -1666.608,E2 -1666.608} C_VEL
LIN {X 0,Y 580.304,Z 512.193,A -85,B 0,C 180,E1 -1669.157,E2 -1669.157} C_VEL
LIN {X 0,Y 580.295,Z 512.195,A -85,B 0,C 180,E1 -1671.927,E2 -1671.927} C_VEL
LIN {X 0,Y 580.256,Z 512.208,A -85,B 0,C 180,E1 -1674.452,E2 -1674.452} C_VEL
LIN {X 0,Y 580.296,Z 512.199,A -85,B 0,C 180,E1 -1676.975,E2 -1676.975} C_VEL
LIN {X 0,Y 580.302,Z 512.195,A -85,B 0,C 180,E1 -1679.425,E2 -1679.425} C_VEL
LIN {X 0,Y 580.302,Z 512.197,A -85,B 0,C 180,E1 -1682.141,E2 -1682.141} C_VEL
LIN {X 0,Y 580.327,Z 512.192,A -85,B 0,C 180,E1 -1685.269,E2 -1685.269} C_VEL
LIN {X 0,Y 580.276,Z 512.198,A -85,B 0,C 180,E1 -1687.947,E2 -1687.947} C_VEL
LIN {X 0,Y 580.35,Z 512.325,A -85,B 0,C 180,E1 -1690.353,E2 -1690.353} C_VEL
LIN {X 0,Y 580.525,Z 518.548,A -85,B 0,C 180,E1 -1691.47,E2 -1691.47} C_VEL
LIN {X 0,Y 580.419,Z 535.32,A -85,B 0,C 180,E1 -1694.37,E2 -1694.37} C_VEL
LIN {X 0,Y 580.353,Z 547.179,A -85,B 0,C 180,E1 -1696.363,E2 -1696.363} C_VEL
LIN {X 0,Y 580.832,Z 550.201,A -85,B 0,C 180,E1 -1696.448,E2 -1696.448} C_VEL
LIN {X 0,Y 580.819,Z 653.884,A -85,B 0,C 180,E1 -1697.752,E2 -1697.752} C_VEL
LIN {X 0,Y 580.757,Z 667.179,A -85,B 0,C 180,E1 -1698.061,E2 -1698.061} C_VEL
LIN {X 0,Y 580.678,Z 679.343,A -85,B 0,C 180,E1 -1698.48,E2 -1698.48} C_VEL
LIN {X 0,Y 580.573,Z 690.777,A -85,B 0,C 180,E1 -1699.008,E2 -1699.008} C_VEL
LIN {X 0,Y 580.456,Z 702.539,A -85,B 0,C 180,E1 -1699.712,E2 -1699.712} C_VEL
LIN {X 0,Y 580.345,Z 713.049,A -85,B 0,C 180,E1 -1700.502,E2 -1700.502} C_VEL
LIN {X 0,Y 580.273,Z 721.652,A -85,B 0,C 180,E1 -1701.292,E2 -1701.292} C_VEL
LIN {X 0,Y 580.222,Z 729.578,A -85,B 0,C 180,E1 -1702.168,E2 -1702.168} C_VEL
LIN {X 0,Y 580.168,Z 737.28,A -85,B 0,C 180,E1 -1703.209,E2 -1703.209} C_VEL
LIN {X 0,Y 580.165,Z 742.618,A -85,B 0,C 180,E1 -1704.089,E2 -1704.089} C_VEL
LIN {X 0,Y 580.053,Z 747.758,A -85,B 0,C 180,E1 -1705.134,E2 -1705.134} C_VEL
LIN {X 0,Y 580.11,Z 751.747,A -85,B 0,C 180,E1 -1706.179,E2 -1706.179} C_VEL
LIN {X 0,Y 580.043,Z 754.697,A -85,B 0,C 180,E1 -1707.221,E2 -1707.221} C_VEL
LIN {X 0,Y 580.039,Z 756.127,A -85,B 0,C 180,E1 -1707.916,E2 -1707.916} C_VEL
LIN {X 0,Y 580.041,Z 757.754,A -85,B 0,C 180,E1 -1709.305,E2 -1709.305} C_VEL
LIN {X 0,Y 580.038,Z 757.996,A -85,B 0,C 180,E1 -1709.999,E2 -1709.999} C_VEL
LIN {X 0,Y 580.04,Z 757.815,A -85,B 0,C 180,E1 -1710.694,E2 -1710.694} C_VEL
LIN {X 0,Y 580.04,Z 756.275,A -85,B 0,C 180,E1 -1712.082,E2 -1712.082} C_VEL
LIN {X 0,Y 580.044,Z 754.914,A -85,B 0,C 180,E1 -1712.777,E2 -1712.777} C_VEL
LIN {X 0,Y 580.11,Z 752.036,A -85,B 0,C 180,E1 -1713.82,E2 -1713.82} C_VEL
LIN {X 0,Y 580.053,Z 748.136,A -85,B 0,C 180,E1 -1714.865,E2 -1714.865} C_VEL
LIN {X 0,Y 580.162,Z 743.105,A -85,B 0,C 180,E1 -1715.909,E2 -1715.909} C_VEL
LIN {X 0,Y 580.157,Z 736.785,A -85,B 0,C 180,E1 -1716.957,E2 -1716.957} C_VEL
LIN {X 0,Y 580.242,Z 728.865,A -85,B 0,C 180,E1 -1718.006,E2 -1718.006} C_VEL
LIN {X 0,Y 580.308,Z 719.018,A -85,B 0,C 180,E1 -1719.058,E2 -1719.058} C_VEL
LIN {X 0,Y 580.418,Z 708.7,A -85,B 0,C 180,E1 -1719.935,E2 -1719.935} C_VEL
LIN {X 0,Y 580.497,Z 698.495,A -85,B 0,C 180,E1 -1720.639,E2 -1720.639} C_VEL
LIN {X 0,Y 580.627,Z 686.166,A -85,B 0,C 180,E1 -1721.312,E2 -1721.312} C_VEL
LIN {X 0,Y 580.704,Z 673.519,A -85,B 0,C 180,E1 -1721.828,E2 -1721.828} C_VEL
LIN {X 0,Y 580.781,Z 660.499,A -85,B 0,C 180,E1 -1722.203,E2 -1722.203} C_VEL
LIN {X 0,Y 580.832,Z 648.183,A -85,B 0,C 180,E1 -1722.424,E2 -1722.424} C_VEL
LIN {X 0,Y 580.812,Z 550.259,A -85,B 0,C 180,E1 -1723.642,E2 -1723.642} C_VEL
LIN {X 0,Y 580.346,Z 547.205,A -85,B 0,C 180,E1 -1723.725,E2 -1723.725} C_VEL
LIN {X 0,Y 580.42,Z 532.705,A -85,B 0,C 180,E1 -1726.17,E2 -1726.17} C_VEL
LIN {X 0,Y 580.544,Z 516.974,A -85,B 0,C 180,E1 -1728.894,E2 -1728.894} C_VEL
LIN {X 0,Y 580.334,Z 512.285,A -85,B 0,C 180,E1 -1729.755,E2 -1729.755} C_VEL
LIN {X 0,Y 580.296,Z 512.198,A -85,B 0,C 180,E1 -1732.802,E2 -1732.802} C_VEL
LIN {X 0,Y 580.308,Z 512.199,A -85,B 0,C 180,E1 -1735.079,E2 -1735.079} C_VEL
LIN {X 0,Y 580.301,Z 512.195,A -85,B 0,C 180,E1 -1738.185,E2 -1738.185} C_VEL
LIN {X 0,Y 580.293,Z 512.196,A -85,B 0,C 180,E1 -1740.695,E2 -1740.695} C_VEL
LIN {X 0,Y 580.304,Z 512.203,A -85,B 0,C 180,E1 -1743.316,E2 -1743.316} C_VEL
LIN {X 0,Y 580.323,Z 512.195,A -85,B 0,C 180,E1 -1745.766,E2 -1745.766} C_VEL
LIN {X 0,Y 580.288,Z 512.197,A -85,B 0,C 180,E1 -1748.145,E2 -1748.145} C_VEL
LIN {X 0,Y 580.299,Z 512.195,A -85,B 0,C 180,E1 -1750.842,E2 -1750.842} C_VEL
LIN {X 0,Y 580.285,Z 512.201,A -85,B 0,C 180,E1 -1753.656,E2 -1753.656} C_VEL
LIN {X 0,Y 580.273,Z 512.197,A -85,B 0,C 180,E1 -1756.608,E2 -1756.608} C_VEL
LIN {X 0,Y 580.301,Z 512.2,A -85,B 0,C 180,E1 -1759.156,E2 -1759.156} C_VEL
LIN {X 0,Y 580.286,Z 512.197,A -85,B 0,C 180,E1 -1761.926,E2 -1761.926} C_VEL
LIN {X 0,Y 580.304,Z 512.194,A -85,B 0,C 180,E1 -1764.456,E2 -1764.456} C_VEL
LIN {X 0,Y 580.288,Z 512.198,A -85,B 0,C 180,E1 -1766.975,E2 -1766.975} C_VEL
LIN {X 0,Y 580.304,Z 512.203,A -85,B 0,C 180,E1 -1769.425,E2 -1769.425} C_VEL
LIN {X 0,Y 580.315,Z 512.193,A -85,B 0,C 180,E1 -1772.136,E2 -1772.136} C_VEL
LIN {X 0,Y 580.304,Z 512.196,A -85,B 0,C 180,E1 -1774.92,E2 -1774.92} C_VEL
LIN {X 0,Y 580.269,Z 512.201,A -85,B 0,C 180,E1 -1777.947,E2 -1777.947} C_VEL
LIN {X 0,Y 580.311,Z 512.194,A -85,B 0,C 180,E1 -1780.914,E2 -1780.914} C_VEL
LIN {X 0,Y 580.276,Z 512.201,A -85,B 0,C 180,E1 -1783.825,E2 -1783.825} C_VEL
LIN {X 0,Y 580.319,Z 512.195,A -85,B 0,C 180,E1 -1785.983,E2 -1785.983} C_VEL
LIN {X 0,Y 580.296,Z 512.195,A -85,B 0,C 180,E1 -1788.827,E2 -1788.827} C_VEL
LIN {X 0,Y 580.329,Z 512.199,A -85,B 0,C 180,E1 -1791.644,E2 -1791.644} C_VEL
LIN {X 0,Y 580.318,Z 512.192,A -85,B 0,C 180,E1 -1794.44,E2 -1794.44} C_VEL
LIN {X 0,Y 580.34,Z 512.193,A -85,B 0,C 180,E1 -1797.223,E2 -1797.223} C_VEL
LIN {X 0,Y 580.345,Z 512.192,A -85,B 0,C 180,E1 -1800,E2 -1800} C_VEL
LIN {X 0,Y 580.34,Z 512.189,A -85,B 0,C 180,E1 -1802.777,E2 -1802.777} C_VEL
LIN {X 0,Y 580.316,Z 512.202,A -85,B 0,C 180,E1 -1805.56,E2 -1805.56} C_VEL
LIN {X 0,Y 580.329,Z 512.191,A -85,B 0,C 180,E1 -1808.356,E2 -1808.356} C_VEL
LIN {X 0,Y 580.292,Z 512.198,A -85,B 0,C 180,E1 -1811.191,E2 -1811.191} C_VEL
LIN {X 0,Y 580.319,Z 512.195,A -85,B 0,C 180,E1 -1814.017,E2 -1814.017} C_VEL
LIN {X 0,Y 580.305,Z 512.194,A -85,B 0,C 180,E1 -1816.914,E2 -1816.914} C_VEL
LIN {X 0,Y 580.3,Z 512.201,A -85,B 0,C 180,E1 -1819.823,E2 -1819.823} C_VEL
LIN {X 0,Y 580.267,Z 512.201,A -85,B 0,C 180,E1 -1822.053,E2 -1822.053} C_VEL
LIN {X 0,Y 580.303,Z 512.196,A -85,B 0,C 180,E1 -1825.08,E2 -1825.08} C_VEL
LIN {X 0,Y 580.314,Z 512.199,A -85,B 0,C 180,E1 -1827.864,E2 -1827.864} C_VEL
LIN {X 0,Y 580.286,Z 512.195,A -85,B 0,C 180,E1 -1830.697,E2 -1830.697} C_VEL
LIN {X 0,Y 580.299,Z 512.199,A -85,B 0,C 180,E1 -1833.317,E2 -1833.317} C_VEL
LIN {X 0,Y 580.322,Z 512.198,A -85,B 0,C 180,E1 -1835.768,E2 -1835.768} C_VEL
LIN {X 0,Y 580.283,Z 512.199,A -85,B 0,C 180,E1 -1838.147,E2 -1838.147} C_VEL
LIN {X 0,Y 580.295,Z 512.195,A -85,B 0,C 180,E1 -1840.844,E2 -1840.844} C_VEL
LIN {X 0,Y 580.274,Z 512.207,A -85,B 0,C 180,E1 -1843.658,E2 -1843.658} C_VEL
LIN {X 0,Y 580.289,Z 512.195,A -85,B 0,C 180,E1 -1846.608,E2 -1846.608} C_VEL
LIN {X 0,Y 580.298,Z 512.197,A -85,B 0,C 180,E1 -1849.158,E2 -1849.158} C_VEL
LIN {X 0,Y 580.289,Z 512.2,A -85,B 0,C 180,E1 -1851.928,E2 -1851.928} C_VEL
LIN {X 0,Y 580.283,Z 512.197,A -85,B 0,C 180,E1 -1854.456,E2 -1854.456} C_VEL
LIN {X 0,Y 580.29,Z 512.195,A -85,B 0,C 180,E1 -1856.976,E2 -1856.976} C_VEL
LIN {X 0,Y 580.302,Z 512.19,A -85,B 0,C 180,E1 -1859.426,E2 -1859.426} C_VEL
LIN {X 0,Y 580.319,Z 512.195,A -85,B 0,C 180,E1 -1862.138,E2 -1862.138} C_VEL
LIN {X 0,Y 580.322,Z 512.196,A -85,B 0,C 180,E1 -1865.27,E2 -1865.27} C_VEL
LIN {X 0,Y 580.306,Z 512.352,A -85,B 0,C 180,E1 -1867.075,E2 -1867.075} C_VEL
LIN {X 0,Y 580.921,Z 516.767,A -85,B 0,C 180,E1 -1867.787,E2 -1867.787} C_VEL
LIN {X 0,Y 580.705,Z 536.848,A -85,B 0,C 180,E1 -1870.735,E2 -1870.735} C_VEL
LIN {X 0,Y 580.524,Z 555.806,A -85,B 0,C 180,E1 -1873.472,E2 -1873.472} C_VEL
LIN {X 0,Y 580.39,Z 575.728,A -85,B 0,C 180,E1 -1876.298,E2 -1876.298} C_VEL
LIN {X 0,Y 580.549,Z 577.127,A -85,B 0,C 180,E1 -1876.358,E2 -1876.358} C_VEL
LIN {X 0,Y 580.956,Z 581.568,A -85,B 0,C 180,E1 -1876.423,E2 -1876.423} C_VEL
LIN {X 0,Y 580.806,Z 683.983,A -85,B 0,C 180,E1 -1877.709,E2 -1877.709} C_VEL
LIN {X 0,Y 580.737,Z 697.239,A -85,B 0,C 180,E1 -1878.018,E2 -1878.018} C_VEL
LIN {X 0,Y 580.677,Z 710.508,A -85,B 0,C 180,E1 -1878.482,E2 -1878.482} C_VEL
LIN {X 0,Y 580.564,Z 721.644,A -85,B 0,C 180,E1 -1879.009,E2 -1879.009} C_VEL
LIN {X 0,Y 580.443,Z 733.212,A -85,B 0,C 180,E1 -1879.713,E2 -1879.713} C_VEL
LIN {X 0,Y 580.341,Z 743.606,A -85,B 0,C 180,E1 -1880.503,E2 -1880.503} C_VEL
LIN {X 0,Y 580.271,Z 752.119,A -85,B 0,C 180,E1 -1881.293,E2 -1881.293} C_VEL
LIN {X 0,Y 580.221,Z 759.966,A -85,B 0,C 180,E1 -1882.169,E2 -1882.169} C_VEL
LIN {X 0,Y 580.153,Z 767.654,A -85,B 0,C 180,E1 -1883.222,E2 -1883.222} C_VEL
LIN {X 0,Y 580.139,Z 774.683,A -85,B 0,C 180,E1 -1884.439,E2 -1884.439} C_VEL
LIN {X 0,Y 580.108,Z 779.374,A -85,B 0,C 180,E1 -1885.484,E2 -1885.484} C_VEL
LIN {X 0,Y 580.123,Z 782.96,A -85,B 0,C 180,E1 -1886.528,E2 -1886.528} C_VEL
LIN {X 0,Y 580.043,Z 784.811,A -85,B 0,C 180,E1 -1887.223,E2 -1887.223} C_VEL
LIN {X 0,Y 580.038,Z 786.202,A -85,B 0,C 180,E1 -1887.918,E2 -1887.918} C_VEL
LIN {X 0,Y 580.04,Z 787.785,A -85,B 0,C 180,E1 -1889.306,E2 -1889.306} C_VEL
LIN {X 0,Y 580.037,Z 788,A -85,B 0,C 180,E1 -1890.001,E2 -1890.001} C_VEL
LIN {X 0,Y 580.047,Z 787.184,A -85,B 0,C 180,E1 -1891.389,E2 -1891.389} C_VEL
LIN {X 0,Y 580.038,Z 786.199,A -85,B 0,C 180,E1 -1892.084,E2 -1892.084} C_VEL
LIN {X 0,Y 580.043,Z 784.807,A -85,B 0,C 180,E1 -1892.779,E2 -1892.779} C_VEL
LIN {X 0,Y 580.109,Z 781.894,A -85,B 0,C 180,E1 -1893.821,E2 -1893.821} C_VEL
LIN {X 0,Y 580.054,Z 777.947,A -85,B 0,C 180,E1 -1894.866,E2 -1894.866} C_VEL
LIN {X 0,Y 580.139,Z 771.874,A -85,B 0,C 180,E1 -1896.085,E2 -1896.085} C_VEL
LIN {X 0,Y 580.185,Z 765.233,A -85,B 0,C 180,E1 -1897.133,E2 -1897.133} C_VEL
LIN {X 0,Y 580.251,Z 756.985,A -85,B 0,C 180,E1 -1898.182,E2 -1898.182} C_VEL
LIN {X 0,Y 580.308,Z 748.532,A -85,B 0,C 180,E1 -1899.059,E2 -1899.059} C_VEL
LIN {X 0,Y 580.415,Z 738.089,A -85,B 0,C 180,E1 -1899.937,E2 -1899.937} C_VEL
LIN {X 0,Y 580.496,Z 727.747,A -85,B 0,C 180,E1 -1900.64,E2 -1900.64} C_VEL
LIN {X 0,Y 580.598,Z 716.224,A -85,B 0,C 180,E1 -1901.265,E2 -1901.265} C_VEL
LIN {X 0,Y 580.681,Z 703.46,A -85,B 0,C 180,E1 -1901.785,E2 -1901.785} C_VEL
LIN {X 0,Y 580.779,Z 690.416,A -85,B 0,C 180,E1 -1902.16,E2 -1902.16} C_VEL
LIN {X 0,Y 580.84,Z 678.043,A -85,B 0,C 180,E1 -1902.38,E2 -1902.38} C_VEL
LIN {X 0,Y 580.875,Z 579.006,A -85,B 0,C 180,E1 -1903.611,E2 -1903.611} C_VEL
LIN {X 0,Y 580.394,Z 575.999,A -85,B 0,C 180,E1 -1903.681,E2 -1903.681} C_VEL
LIN {X 0,Y 580.525,Z 557.056,A -85,B 0,C 180,E1 -1906.349,E2 -1906.349} C_VEL
LIN {X 0,Y 580.695,Z 538.166,A -85,B 0,C 180,E1 -1909.074,E2 -1909.074} C_VEL
LIN {X 0,Y 580.903,Z 519.278,A -85,B 0,C 180,E1 -1911.841,E2 -1911.841} C_VEL
LIN {X 0,Y 580.673,Z 514.239,A -85,B 0,C 180,E1 -1912.599,E2 -1912.599} C_VEL
LIN {X 0,Y 580.307,Z 512.344,A -85,B 0,C 180,E1 -1912.926,E2 -1912.926} C_VEL
LIN {X 0,Y 580.309,Z 512.195,A -85,B 0,C 180,E1 -1915.08,E2 -1915.08} C_VEL
LIN {X 0,Y 580.302,Z 512.201,A -85,B 0,C 180,E1 -1918.186,E2 -1918.186} C_VEL
LIN {X 0,Y 580.288,Z 512.199,A -85,B 0,C 180,E1 -1920.695,E2 -1920.695} C_VEL
LIN {X 0,Y 580.306,Z 512.195,A -85,B 0,C 180,E1 -1923.316,E2 -1923.316} C_VEL
LIN {X 0,Y 580.248,Z 512.206,A -85,B 0,C 180,E1 -1925.756,E2 -1925.756} C_VEL
LIN {X 0,Y 580.293,Z 512.204,A -85,B 0,C 180,E1 -1928.146,E2 -1928.146} C_VEL
LIN {X 0,Y 580.302,Z 512.195,A -85,B 0,C 180,E1 -1930.844,E2 -1930.844} C_VEL
LIN {X 0,Y 580.293,Z 512.2,A -85,B 0,C 180,E1 -1933.657,E2 -1933.657} C_VEL
LIN {X 0,Y 580.28,Z 512.199,A -85,B 0,C 180,E1 -1936.609,E2 -1936.609} C_VEL
LIN {X 0,Y 580.303,Z 512.195,A -85,B 0,C 180,E1 -1939.157,E2 -1939.157} C_VEL
LIN {X 0,Y 580.294,Z 512.205,A -85,B 0,C 180,E1 -1941.927,E2 -1941.927} C_VEL
LIN {X 0,Y 580.31,Z 512.195,A -85,B 0,C 180,E1 -1944.457,E2 -1944.457} C_VEL
LIN {X 0,Y 580.295,Z 512.196,A -85,B 0,C 180,E1 -1946.975,E2 -1946.975} C_VEL
LIN {X 0,Y 580.299,Z 512.2,A -85,B 0,C 180,E1 -1949.425,E2 -1949.425} C_VEL
LIN {X 0,Y 580.296,Z 512.201,A -85,B 0,C 180,E1 -1952.142,E2 -1952.142} C_VEL
LIN {X 0,Y 580.335,Z 512.419,A -85,B 0,C 180,E1 -1954.874,E2 -1954.874} C_VEL
LIN {X 0,Y 581.182,Z 516.805,A -85,B 0,C 180,E1 -1955.527,E2 -1955.527} C_VEL
LIN {X 0,Y 581.071,Z 532.472,A -85,B 0,C 180,E1 -1957.605,E2 -1957.605} C_VEL
LIN {X 0,Y 580.828,Z 554.823,A -85,B 0,C 180,E1 -1960.515,E2 -1960.515} C_VEL
LIN {X 0,Y 580.614,Z 576.51,A -85,B 0,C 180,E1 -1963.293,E2 -1963.293} C_VEL
LIN {X 0,Y 580.489,Z 599.241,A -85,B 0,C 180,E1 -1966.166,E2 -1966.166} C_VEL
LIN {X 0,Y 580.34,Z 624.928,A -85,B 0,C 180,E1 -1969.372,E2 -1969.372} C_VEL
LIN {X 0,Y 580.317,Z 630.968,A -85,B 0,C 180,E1 -1970.106,E2 -1970.106} C_VEL
LIN {X 0,Y 580.537,Z 635.934,A -85,B 0,C 180,E1 -1970.198,E2 -1970.198} C_VEL
LIN {X 0,Y 580.492,Z 702.26,A -85,B 0,C 180,E1 -1971.032,E2 -1971.032} C_VEL
LIN {X 0,Y 580.446,Z 713.016,A -85,B 0,C 180,E1 -1971.295,E2 -1971.295} C_VEL
LIN {X 0,Y 580.388,Z 722.436,A -85,B 0,C 180,E1 -1971.645,E2 -1971.645} C_VEL
LIN {X 0,Y 580.334,Z 732.661,A -85,B 0,C 180,E1 -1972.17,E2 -1972.17} C_VEL
LIN {X 0,Y 580.261,Z 741.801,A -85,B 0,C 180,E1 -1972.781,E2 -1972.781} C_VEL
LIN {X 0,Y 580.204,Z 750.891,A -85,B 0,C 180,E1 -1973.576,E2 -1973.576} C_VEL
LIN {X 0,Y 580.174,Z 757.149,A -85,B 0,C 180,E1 -1974.264,E2 -1974.264} C_VEL
LIN {X 0,Y 580.131,Z 763.515,A -85,B 0,C 180,E1 -1975.135,E2 -1975.135} C_VEL
LIN {X 0,Y 580.139,Z 769.299,A -85,B 0,C 180,E1 -1976.18,E2 -1976.18} C_VEL
LIN {X 0,Y 580.055,Z 773.427,A -85,B 0,C 180,E1 -1977.222,E2 -1977.222} C_VEL
LIN {X 0,Y 580.035,Z 775.403,A -85,B 0,C 180,E1 -1977.917,E2 -1977.917} C_VEL
LIN {X 0,Y 580.042,Z 776.833,A -85,B 0,C 180,E1 -1978.611,E2 -1978.611} C_VEL
LIN {X 0,Y 580.035,Z 777.691,A -85,B 0,C 180,E1 -1979.306,E2 -1979.306} C_VEL
